C03619=1103.138,282.672,422.520,179.278,15.807,151.492
C03620=1103.132,282.424,422.550,179.274,15.805,151.492
C03621=1103.126,282.176,422.578,179.271,15.805,151.493
C03622=1103.121,281.927,422.607,179.267,15.803,151.493
C03623=1103.115,281.679,422.636,179.264,15.802,151.494
C03624=1103.109,281.431,422.666,179.260,15.801,151.494
C03625=1103.104,281.183,422.695,179.256,15.800,151.495
C03626=1103.098,280.935,422.724,179.252,15.799,151.495
C03627=1103.092,280.687,422.753,179.249,15.798,151.496
C03628=1103.087,280.438,422.782,179.245,15.797,151.496
C03629=1103.081,280.190,422.811,179.242,15.796,151.497
C03630=1103.076,279.942,422.841,179.238,15.795,151.497
C03631=1103.069,279.694,422.870,179.235,15.794,151.498
C03632=1103.064,279.446,422.899,179.231,15.793,151.498
C03633=1103.059,279.197,422.927,179.227,15.792,151.499
C03634=1103.053,278.949,422.957,179.224,15.791,151.499
C03635=1103.047,278.701,422.986,179.220,15.790,151.500
C03636=1103.041,278.453,423.014,179.216,15.789,151.500
C03637=1103.036,278.204,423.044,179.212,15.788,151.501
C03638=1103.030,277.956,423.073,179.209,15.787,151.502
C03639=1103.025,277.708,423.101,179.205,15.786,151.502
C03640=1103.019,277.460,423.130,179.202,15.785,151.503
C03641=1103.013,277.211,423.159,179.198,15.784,151.503
C03642=1103.008,276.963,423.188,179.195,15.783,151.504
C03643=1103.000,276.606,423.229,179.189,15.782,151.504
C03644=1102.991,276.250,423.271,179.184,15.781,151.505
C03645=1102.984,275.893,423.312,179.179,15.780,151.506
C03646=1102.975,275.536,423.353,179.174,15.778,151.507
C03647=1102.969,275.288,423.382,179.170,15.777,151.507
C03648=1102.964,275.039,423.411,179.167,15.776,151.508
C03649=1102.958,274.791,423.440,179.163,15.775,151.508
C03650=1102.952,274.543,423.468,179.159,15.774,151.509
C03651=1102.946,274.294,423.497,179.155,15.773,151.509
C03652=1102.941,274.046,423.526,179.152,15.772,151.510
C03653=1102.935,273.797,423.554,179.148,15.771,151.511
C03654=1102.930,273.550,423.583,179.145,15.770,151.511
C03655=1102.924,273.301,423.611,179.141,15.769,151.512
C03656=1102.918,273.053,423.641,179.138,15.769,151.512
C03657=1102.913,272.805,423.669,179.134,15.767,151.513
C03658=1102.907,272.556,423.697,179.130,15.767,151.513
C03659=1102.901,272.308,423.726,179.127,15.766,151.514
C03660=1102.896,272.060,423.754,179.123,15.765,151.515
C03661=1102.891,271.811,423.783,179.120,15.764,151.515
C03662=1102.885,271.563,423.812,179.116,15.763,151.516
C03663=1102.879,271.314,423.840,179.112,15.762,151.516
C03664=1102.873,271.066,423.868,179.108,15.762,151.517
C03665=1102.867,270.818,423.897,179.105,15.761,151.517
C03666=1102.862,270.570,423.925,179.101,15.760,151.518
C03667=1102.856,270.321,423.953,179.098,15.759,151.518
C03668=1102.851,270.073,423.981,179.094,15.758,151.519
C03669=1102.845,269.825,424.011,179.090,15.757,151.520
C03670=1102.840,269.577,424.039,179.086,15.756,151.520
C03671=1102.834,269.328,424.067,179.083,15.756,151.521
C03672=1102.828,269.079,424.096,179.080,15.755,151.521
C03673=1102.822,268.831,424.124,179.076,15.754,151.522
C03674=1102.816,268.583,424.152,179.072,15.753,151.522
C03675=1102.811,268.335,424.181,179.068,15.752,151.523
C03676=1102.805,268.086,424.209,179.065,15.751,151.524
C03677=1102.800,267.838,424.237,179.061,15.750,151.524
C03678=1102.794,267.590,424.265,179.057,15.750,151.525
C03679=1102.788,267.342,424.293,179.054,15.749,151.525
C03680=1102.782,267.093,424.321,179.050,15.748,151.526
C03681=1102.777,266.845,424.349,179.047,15.748,151.527
C03682=1102.771,266.596,424.378,179.043,15.746,151.527
C03683=1102.766,266.348,424.406,179.040,15.746,151.528
C03684=1102.760,266.100,424.434,179.035,15.745,151.528
C03685=1102.754,265.851,424.462,179.032,15.744,151.529
C03686=1102.749,265.603,424.490,179.028,15.743,151.529
C03687=1102.743,265.354,424.518,179.025,15.743,151.530
C03688=1102.738,265.106,424.546,179.021,15.742,151.531
C03689=1102.732,264.858,424.575,179.017,15.741,151.531
C03690=1102.726,264.610,424.602,179.014,15.740,151.532
C03691=1102.720,264.362,424.630,179.010,15.739,151.532
C03692=1102.714,264.113,424.658,179.006,15.739,151.533
C03693=1102.709,263.865,424.686,179.003,15.738,151.534
C03694=1102.703,263.616,424.714,178.999,15.737,151.534
C03695=1102.695,263.263,424.754,178.994,15.736,151.535
C03696=1102.686,262.908,424.793,178.988,15.735,151.536
C03697=1102.679,262.554,424.833,178.984,15.735,151.537
C03698=1102.670,262.200,424.873,178.978,15.733,151.538
C03699=1102.665,261.952,424.901,178.974,15.732,151.538
C03700=1102.659,261.703,424.929,178.971,15.732,151.539
C03701=1102.653,261.455,424.956,178.968,15.731,151.539
C03702=1102.647,261.206,424.984,178.963,15.730,151.540
C03703=1102.642,260.958,425.012,178.960,15.730,151.541
C03704=1102.636,260.710,425.040,178.956,15.729,151.541
C03705=1102.630,260.461,425.067,178.953,15.728,151.542
C03706=1102.625,260.213,425.095,178.949,15.728,151.543
C03707=1102.618,259.964,425.123,178.945,15.727,151.543
C03708=1102.613,259.716,425.150,178.941,15.726,151.544
C03709=1102.608,259.468,425.178,178.938,15.726,151.544
C03710=1102.601,259.219,425.206,178.934,15.725,151.545
C03711=1102.596,258.971,425.233,178.931,15.724,151.546
C03712=1102.591,258.723,425.261,178.926,15.723,151.546
C03713=1102.584,258.474,425.289,178.923,15.723,151.547
C03714=1102.579,258.225,425.316,178.920,15.722,151.548
C03715=1102.573,257.977,425.344,178.915,15.721,151.548
C03716=1102.567,257.728,425.371,178.912,15.721,151.549
C03717=1102.562,257.480,425.399,178.909,15.721,151.549
C03718=1102.556,257.233,425.426,178.905,15.719,151.550
C03719=1102.550,256.983,425.454,178.901,15.719,151.551
C03720=1102.545,256.735,425.482,178.898,15.718,151.551
C03721=1102.539,256.487,425.509,178.894,15.717,151.552
C03722=1102.533,256.238,425.537,178.890,15.717,151.552
C03723=1102.527,255.990,425.564,178.886,15.716,151.553
C03724=1102.522,255.742,425.591,178.883,15.715,151.554
C03725=1102.517,255.493,425.619,178.879,15.715,151.554
C03726=1102.510,255.244,425.646,178.875,15.714,151.555
C03727=1102.505,254.996,425.674,178.872,15.714,151.556
C03728=1102.499,254.747,425.700,178.868,15.713,151.556
C03729=1102.494,254.499,425.728,178.864,15.712,151.557
C03730=1102.488,254.250,425.755,178.861,15.712,151.558
C03731=1102.483,254.002,425.783,178.858,15.711,151.558
C03732=1102.476,253.754,425.810,178.853,15.710,151.559
C03733=1102.471,253.505,425.837,178.850,15.710,151.559
C03734=1102.465,253.257,425.865,178.847,15.709,151.560
C03735=1102.460,253.008,425.892,178.843,15.708,151.561
C03736=1102.454,252.760,425.919,178.839,15.708,151.561
C03737=1102.449,252.511,425.946,178.835,15.707,151.562
C03738=1102.443,252.263,425.973,178.832,15.706,151.562
C03739=1102.438,252.015,426.001,178.828,15.706,151.563
C03740=1102.431,251.766,426.028,178.824,15.705,151.564
C03741=1102.426,251.517,426.055,178.821,15.705,151.564
C03742=1102.420,251.269,426.082,178.817,15.704,151.565
C03743=1102.415,251.021,426.109,178.813,15.703,151.566
C03744=1102.410,250.772,426.136,178.810,15.702,151.566
C03745=1102.404,250.524,426.163,178.806,15.702,151.567
C03746=1102.398,250.274,426.190,178.802,15.701,151.568
C03747=1102.390,249.918,426.230,178.797,15.701,151.568
C03748=1102.382,249.561,426.268,178.792,15.700,151.569
C03749=1102.374,249.204,426.307,178.787,15.699,151.570
C03750=1102.366,248.847,426.347,178.781,15.698,151.571
C03751=1102.361,248.599,426.373,178.778,15.697,151.572
C03752=1102.355,248.351,426.400,178.775,15.697,151.572
C03753=1102.350,248.102,426.427,178.770,15.696,151.573
C03754=1102.344,247.854,426.454,178.767,15.695,151.574
C03755=1102.339,247.605,426.481,178.764,15.695,151.574
C03756=1102.333,247.357,426.508,178.760,15.694,151.575
C03757=1102.327,247.108,426.534,178.756,15.694,151.575
C03758=1102.322,246.860,426.561,178.753,15.693,151.576
C03759=1102.317,246.611,426.588,178.749,15.692,151.577
C03760=1102.311,246.363,426.615,178.745,15.692,151.577
C03761=1102.304,246.114,426.642,178.741,15.692,151.578
C03762=1102.299,245.865,426.668,178.738,15.691,151.579
C03763=1102.294,245.617,426.696,178.734,15.690,151.579
C03764=1102.288,245.368,426.722,178.730,15.690,151.580
C03765=1102.282,245.120,426.749,178.727,15.689,151.581
C03766=1102.276,244.872,426.776,178.723,15.688,151.581
C03767=1102.272,244.622,426.802,178.719,15.688,151.582
C03768=1102.266,244.374,426.829,178.716,15.688,151.583
C03769=1102.260,244.126,426.855,178.713,15.687,151.583
C03770=1102.254,243.877,426.882,178.708,15.687,151.584
C03771=1102.248,243.629,426.909,178.705,15.686,151.584
C03772=1102.243,243.381,426.935,178.702,15.686,151.585
C03773=1102.238,243.131,426.962,178.697,15.685,151.586
C03774=1102.232,242.883,426.989,178.694,15.684,151.586
C03775=1102.226,242.635,427.015,178.691,15.684,151.587
C03776=1102.221,242.386,427.042,178.687,15.684,151.588
C03777=1102.215,242.138,427.069,178.683,15.683,151.589
C03778=1102.209,241.889,427.094,178.680,15.682,151.589
C03779=1102.204,241.641,427.121,178.676,15.682,151.590
C03780=1102.198,241.392,427.148,178.672,15.681,151.590
C03781=1102.192,241.144,427.174,178.668,15.681,151.591
C03782=1102.187,240.895,427.200,178.665,15.681,151.592
C03783=1102.181,240.646,427.227,178.661,15.680,151.592
C03784=1102.175,240.398,427.254,178.657,15.679,151.593
C03785=1102.170,240.149,427.280,178.654,15.679,151.594
C03786=1102.164,239.901,427.306,178.650,15.679,151.595
C03787=1102.158,239.652,427.333,178.647,15.678,151.595
C03788=1102.153,239.403,427.359,178.642,15.677,151.596
C03789=1102.147,239.155,427.385,178.639,15.677,151.597
C03790=1102.141,238.906,427.411,178.635,15.677,151.597
C03791=1102.136,238.658,427.438,178.632,15.676,151.598
C03792=1102.130,238.409,427.465,178.628,15.676,151.598
C03793=1102.124,238.160,427.491,178.624,15.675,151.599
C03794=1102.119,237.912,427.517,178.621,15.675,151.600
C03795=1102.113,237.663,427.543,178.617,15.675,151.601
C03796=1102.107,237.415,427.569,178.613,15.674,151.601
C03797=1102.101,237.166,427.595,178.610,15.674,151.602
C03798=1102.095,236.918,427.622,178.606,15.673,151.603
C03799=1102.088,236.554,427.660,178.601,15.672,151.603
C03800=1102.079,236.190,427.698,178.595,15.672,151.604
C03801=1102.071,235.827,427.737,178.591,15.671,151.605
C03802=1102.063,235.463,427.774,178.585,15.671,151.606
C03803=1102.057,235.214,427.801,178.581,15.670,151.607
C03804=1102.052,234.965,427.827,178.578,15.670,151.608
C03805=1102.046,234.718,427.853,178.574,15.669,151.608
C03806=1102.041,234.469,427.879,178.570,15.669,151.609
C03807=1102.035,234.220,427.905,178.567,15.669,151.610
C03808=1102.029,233.972,427.931,178.563,15.668,151.610
C03809=1102.023,233.723,427.957,178.559,15.667,151.611
C03810=1102.018,233.474,427.983,178.556,15.667,151.612
C03811=1102.013,233.226,428.009,178.552,15.667,151.612
C03812=1102.007,232.977,428.034,178.549,15.667,151.613
C03813=1102.001,232.728,428.060,178.545,15.666,151.614
C03814=1101.996,232.479,428.086,178.541,15.666,151.615
C03815=1101.990,232.231,428.113,178.538,15.665,151.615
C03816=1101.984,231.982,428.138,178.534,15.665,151.616
C03817=1101.979,231.734,428.164,178.530,15.665,151.617
C03818=1101.973,231.485,428.190,178.526,15.664,151.617
C03819=1101.968,231.237,428.216,178.523,15.663,151.618
C03820=1101.961,230.988,428.242,178.519,15.663,151.619
C03821=1101.956,230.739,428.268,178.516,15.663,151.619
C03822=1101.951,230.491,428.293,178.512,15.662,151.620
C03823=1101.945,230.242,428.319,178.508,15.662,151.621
C03824=1101.939,229.993,428.345,178.505,15.661,151.621
C03825=1101.933,229.745,428.371,178.501,15.661,151.622
C03826=1101.927,229.496,428.397,178.497,15.661,151.623
C03827=1101.923,229.248,428.422,178.494,15.661,151.623
C03828=1101.916,228.999,428.447,178.491,15.660,151.624
C03829=1101.911,228.750,428.473,178.486,15.659,151.625
C03830=1101.905,228.502,428.499,178.483,15.659,151.625
C03831=1101.900,228.253,428.524,178.479,15.659,151.626
C03832=1101.894,228.005,428.550,178.476,15.659,151.627
C03833=1101.888,227.756,428.576,178.472,15.659,151.628
C03834=1101.882,227.507,428.601,178.468,15.658,151.628
C03835=1101.877,227.259,428.626,178.464,15.658,151.629
C03836=1101.872,227.010,428.652,178.461,15.658,151.630
C03837=1101.865,226.761,428.678,178.458,15.657,151.630
C03838=1101.860,226.512,428.704,178.454,15.657,151.631
C03839=1101.854,226.264,428.729,178.451,15.657,151.632
C03840=1101.849,226.015,428.755,178.446,15.656,151.632
C03841=1101.843,225.766,428.780,178.443,15.656,151.633
C03842=1101.838,225.518,428.806,178.439,15.655,151.634
C03843=1101.832,225.269,428.831,178.436,15.655,151.635
C03844=1101.826,225.020,428.857,178.432,15.655,151.635
C03845=1101.820,224.772,428.882,178.429,15.654,151.636
C03846=1101.815,224.523,428.906,178.425,15.654,151.636
C03847=1101.809,224.274,428.932,178.421,15.653,151.637
C03848=1101.803,224.026,428.958,178.417,15.653,151.638
C03849=1101.798,223.777,428.983,178.414,15.653,151.639
C03850=1101.792,223.529,429.009,178.410,15.653,151.639
C03851=1101.784,223.156,429.046,178.405,15.652,151.640
C03852=1101.776,222.784,429.084,178.399,15.651,151.641
C03853=1101.767,222.412,429.122,178.394,15.651,151.642
C03854=1101.759,222.040,429.160,178.389,15.651,151.643
C03855=1101.753,221.792,429.185,178.385,15.651,151.644
C03856=1101.747,221.543,429.210,178.382,15.650,151.645
C03857=1101.741,221.294,429.236,178.377,15.650,151.646
C03858=1101.737,221.045,429.260,178.374,15.649,151.646
C03859=1101.730,220.797,429.286,178.370,15.649,151.647
C03860=1101.724,220.548,429.311,178.367,15.649,151.648
C03861=1101.719,220.299,429.335,178.363,15.649,151.648
C03862=1101.713,220.050,429.361,178.360,15.649,151.649
C03863=1101.707,219.802,429.387,178.356,15.649,151.650
C03864=1101.702,219.553,429.411,178.352,15.648,151.651
C03865=1101.696,219.304,429.436,178.349,15.647,151.651
C03866=1101.691,219.056,429.461,178.345,15.647,151.652
C03867=1101.685,218.807,429.486,178.341,15.647,151.653
C03868=1101.679,218.559,429.511,178.338,15.647,151.653
C03869=1101.673,218.310,429.536,178.334,15.647,151.654
C03870=1101.668,218.061,429.562,178.331,15.646,151.655
C03871=1101.663,217.812,429.586,178.327,15.646,151.655
C03872=1101.656,217.563,429.612,178.323,15.645,151.656
C03873=1101.651,217.315,429.636,178.319,15.645,151.657
C03874=1101.645,217.066,429.661,178.316,15.645,151.658
C03875=1101.640,216.817,429.686,178.312,15.645,151.658
C03876=1101.634,216.569,429.711,178.309,15.645,151.659
C03877=1101.629,216.320,429.736,178.305,15.645,151.660
C03878=1101.623,216.071,429.761,178.302,15.644,151.660
C03879=1101.617,215.823,429.785,178.298,15.644,151.661
C03880=1101.611,215.574,429.811,178.295,15.644,151.662
C03881=1101.606,215.326,429.835,178.291,15.643,151.662
C03882=1101.601,215.076,429.860,178.287,15.643,151.663
C03883=1101.595,214.828,429.885,178.284,15.643,151.664
C03884=1101.589,214.579,429.910,178.280,15.642,151.665
C03885=1101.584,214.331,429.935,178.276,15.642,151.665
C03886=1101.578,214.081,429.959,178.273,15.642,151.666
C03887=1101.572,213.833,429.983,178.269,15.642,151.667
C03888=1101.567,213.585,430.008,178.266,15.642,151.667
C03889=1101.561,213.336,430.033,178.262,15.642,151.668
C03890=1101.556,213.087,430.057,178.258,15.641,151.669
C03891=1101.550,212.838,430.082,178.254,15.641,151.670
C03892=1101.544,212.590,430.107,178.251,15.641,151.670
C03893=1101.538,212.340,430.131,178.247,15.640,151.671
C03894=1101.533,212.092,430.156,178.244,15.640,151.672
C03895=1101.527,211.843,430.181,178.240,15.640,151.672
C03896=1101.521,211.595,430.205,178.237,15.640,151.673
C03897=1101.516,211.346,430.230,178.233,15.640,151.674
C03898=1101.510,211.097,430.254,178.230,15.639,151.674
C03899=1101.505,210.848,430.278,178.226,15.639,151.675
C03900=1101.499,210.599,430.304,178.223,15.639,151.676
C03901=1101.493,210.351,430.328,178.218,15.638,151.677
C03902=1101.487,210.102,430.353,178.215,15.638,151.677
C03903=1101.480,209.733,430.389,178.210,15.638,151.678
C03904=1101.471,209.366,430.425,178.204,15.637,151.679
C03905=1101.463,208.997,430.461,178.199,15.638,151.680
C03906=1101.455,208.628,430.497,178.194,15.637,151.682
C03907=1101.431,207.624,430.595,178.158,15.629,151.687
C03908=1101.426,207.375,430.619,178.154,15.629,151.688
C03909=1101.420,207.126,430.644,178.150,15.630,151.689
C03910=1101.414,206.878,430.668,178.146,15.630,151.690
C03911=1101.409,206.629,430.692,178.143,15.631,151.691
C03912=1101.403,206.380,430.717,178.139,15.632,151.692
C03913=1101.397,206.132,430.740,178.135,15.632,151.693
C03914=1101.392,205.882,430.764,178.131,15.633,151.694
C03915=1101.387,205.634,430.788,178.128,15.634,151.695
C03916=1101.381,205.384,430.813,178.124,15.634,151.696
C03917=1101.375,205.136,430.836,178.120,15.635,151.697
C03918=1101.369,204.888,430.861,178.116,15.635,151.698
C03919=1101.363,204.638,430.885,178.112,15.636,151.699
C03920=1101.357,204.390,430.909,178.109,15.637,151.700
C03921=1101.352,204.141,430.932,178.105,15.637,151.700
C03922=1101.347,203.892,430.957,178.100,15.638,151.701
C03923=1101.340,203.643,430.981,178.097,15.638,151.702
C03924=1101.335,203.395,431.005,178.094,15.639,151.703
C03925=1101.330,203.145,431.028,178.089,15.640,151.704
C03926=1101.324,202.897,431.052,178.086,15.640,151.705
C03927=1101.319,202.649,431.076,178.082,15.641,151.706
C03928=1101.312,202.400,431.100,178.077,15.641,151.707
C03929=1101.307,202.150,431.124,178.074,15.642,151.708
C03930=1101.301,201.902,431.148,178.070,15.643,151.709
C03931=1101.295,201.653,431.172,178.066,15.643,151.710
C03932=1101.289,201.405,431.196,178.063,15.644,151.711
C03933=1101.284,201.155,431.219,178.059,15.645,151.712
C03934=1101.278,200.907,431.243,178.055,15.645,151.713
C03935=1101.272,200.658,431.268,178.051,15.646,151.714
C03936=1101.267,200.409,431.291,178.047,15.646,151.715
C03937=1101.260,200.161,431.314,178.044,15.647,151.715
C03938=1101.255,199.911,431.338,178.040,15.648,151.717
C03939=1101.249,199.662,431.362,178.036,15.649,151.717
C03940=1101.244,199.414,431.386,178.032,15.649,151.718
C03941=1101.238,199.165,431.409,178.029,15.650,151.719
C03942=1101.233,198.916,431.433,178.025,15.651,151.720
C03943=1101.227,198.668,431.456,178.021,15.651,151.721
C03944=1101.220,198.419,431.480,178.017,15.652,151.722
C03945=1101.215,198.169,431.504,178.014,15.653,151.723
C03946=1101.209,197.921,431.527,178.010,15.653,151.724
C03947=1101.204,197.672,431.551,178.006,15.654,151.725
C03948=1101.198,197.424,431.575,178.002,15.654,151.726
C03949=1101.192,197.175,431.598,177.999,15.655,151.727
C03950=1101.187,196.926,431.622,177.995,15.656,151.728
C03951=1101.181,196.676,431.645,177.991,15.656,151.729
C03952=1101.175,196.428,431.669,177.987,15.656,151.729
C03953=1101.170,196.179,431.692,177.984,15.657,151.730
C03954=1101.164,195.931,431.716,177.980,15.658,151.731
C03955=1101.159,195.682,431.740,177.976,15.658,151.732
C03956=1101.153,195.433,431.763,177.972,15.659,151.733
C03957=1101.147,195.184,431.786,177.969,15.660,151.734
C03958=1101.142,194.935,431.810,177.965,15.660,151.735
C03959=1101.135,194.686,431.834,177.961,15.661,151.736
C03960=1101.130,194.437,431.857,177.957,15.661,151.737
C03961=1101.124,194.188,431.880,177.954,15.662,151.738
C03962=1101.119,193.940,431.904,177.950,15.662,151.739
C03963=1101.113,193.691,431.927,177.946,15.663,151.739
C03964=1101.107,193.442,431.950,177.942,15.663,151.741
C03965=1101.102,193.193,431.974,177.939,15.664,151.741
C03966=1101.096,192.944,431.997,177.935,15.665,151.742
C03967=1101.090,192.696,432.020,177.931,15.665,151.743
C03968=1101.084,192.423,432.046,177.927,15.666,151.744
C03969=1101.079,192.150,432.071,177.923,15.666,151.745
C03970=1101.071,191.877,432.097,177.919,15.667,151.746
C03971=1101.066,191.604,432.122,177.915,15.667,151.747
C03972=1101.059,191.356,432.146,177.911,15.668,151.748
C03973=1101.054,191.107,432.169,177.908,15.669,151.749
C03974=1101.049,190.858,432.192,177.904,15.669,151.750
C03975=1101.043,190.609,432.215,177.900,15.670,151.751
C03976=1101.037,190.360,432.238,177.896,15.670,151.752
C03977=1101.032,190.112,432.262,177.893,15.671,151.753
C03978=1101.026,189.863,432.285,177.889,15.671,151.753
C03979=1101.021,189.614,432.308,177.886,15.672,151.754
C03980=1101.015,189.365,432.331,177.882,15.672,151.755
C03981=1101.010,189.116,432.355,177.879,15.673,151.756
C03982=1101.005,188.868,432.377,177.875,15.673,151.757
C03983=1100.999,188.619,432.400,177.871,15.674,151.758
C03984=1100.993,188.370,432.423,177.867,15.674,151.759
C03985=1100.987,188.121,432.446,177.864,15.675,151.760
C03986=1100.982,187.872,432.469,177.860,15.675,151.760
C03987=1100.977,187.623,432.493,177.856,15.676,151.761
C03988=1100.971,187.374,432.516,177.852,15.676,151.762
C03989=1100.965,187.125,432.539,177.849,15.677,151.763
C03990=1100.959,186.877,432.562,177.845,15.677,151.764
C03991=1100.954,186.627,432.585,177.841,15.678,151.765
C03992=1100.948,186.378,432.607,177.838,15.677,151.766
C03993=1100.943,186.129,432.631,177.835,15.678,151.766
C03994=1100.938,185.881,432.654,177.831,15.679,151.767
C03995=1100.932,185.632,432.677,177.827,15.679,151.768
C03996=1100.927,185.383,432.699,177.824,15.680,151.769
C03997=1100.921,185.134,432.722,177.820,15.680,151.770
C03998=1100.915,184.885,432.745,177.816,15.681,151.771
C03999=1100.909,184.636,432.768,177.812,15.681,151.772
C04000=1100.904,184.387,432.791,177.809,15.682,151.773
C04001=1100.898,184.139,432.814,177.805,15.682,151.774
C04002=1100.891,183.890,432.837,177.802,15.683,151.774
C04003=1100.886,183.641,432.859,177.799,15.684,151.775
C04004=1100.880,183.392,432.882,177.795,15.684,151.776
C04005=1100.875,183.143,432.905,177.791,15.684,151.777
C04006=1100.869,182.894,432.928,177.787,15.685,151.778
C04007=1100.863,182.645,432.951,177.784,15.686,151.779
C04008=1100.857,182.396,432.973,177.780,15.686,151.780
C04009=1100.851,182.147,432.996,177.776,15.687,151.781
C04010=1100.846,181.899,433.018,177.773,15.688,151.781
C04011=1100.840,181.650,433.041,177.769,15.688,151.782
C04012=1100.835,181.401,433.064,177.765,15.688,151.783
C04013=1100.829,181.152,433.087,177.761,15.689,151.784
C04014=1100.822,180.903,433.109,177.758,15.690,151.785
C04015=1100.817,180.654,433.131,177.754,15.690,151.786
C04016=1100.811,180.405,433.154,177.751,15.690,151.787
C04017=1100.805,180.156,433.177,177.748,15.691,151.788
C04018=1100.799,179.907,433.199,177.744,15.692,151.789
C04019=1100.794,179.659,433.221,177.740,15.692,151.789
C04020=1100.788,179.410,433.244,177.737,15.693,151.790
C04021=1100.783,179.161,433.267,177.733,15.693,151.791
C04022=1100.777,178.912,433.289,177.729,15.693,151.792
C04023=1100.771,178.663,433.312,177.725,15.694,151.793
C04024=1100.765,178.414,433.335,177.722,15.695,151.794
C04025=1100.760,178.164,433.357,177.718,15.695,151.795
C04026=1100.754,177.916,433.379,177.715,15.695,151.796
C04027=1100.748,177.667,433.401,177.712,15.696,151.796
C04028=1100.743,177.418,433.424,177.708,15.696,151.797
C04029=1100.737,177.169,433.447,177.704,15.697,151.798
C04030=1100.731,176.920,433.469,177.701,15.698,151.799
C04031=1100.726,176.672,433.491,177.697,15.698,151.800
C04032=1100.719,176.399,433.516,177.693,15.698,151.801
C04033=1100.712,176.125,433.540,177.689,15.699,151.802
C04034=1100.707,175.852,433.565,177.686,15.699,151.802
C04035=1100.701,175.579,433.589,177.681,15.700,151.803
C04036=1100.695,175.331,433.611,177.678,15.700,151.804
C04037=1100.689,175.081,433.634,177.675,15.701,151.805
C04038=1100.684,174.832,433.656,177.671,15.701,151.806
C04039=1100.677,174.583,433.678,177.667,15.702,151.807
C04040=1100.672,174.335,433.701,177.664,15.702,151.808
C04041=1100.667,174.085,433.723,177.660,15.702,151.808
C04042=1100.661,173.836,433.745,177.656,15.703,151.809
C04043=1100.655,173.587,433.768,177.653,15.703,151.810
C04044=1100.650,173.338,433.789,177.650,15.704,151.811
C04045=1100.644,173.090,433.812,177.646,15.704,151.812
C04046=1100.638,172.840,433.834,177.642,15.704,151.813
C04047=1100.633,172.592,433.856,177.639,15.705,151.813
C04048=1100.627,172.343,433.878,177.635,15.705,151.814
C04049=1100.622,172.093,433.900,177.632,15.705,151.815
C04050=1100.616,171.846,433.922,177.629,15.706,151.816
C04051=1100.610,171.596,433.945,177.625,15.706,151.817
C04052=1100.605,171.347,433.967,177.621,15.707,151.818
C04053=1100.599,171.098,433.988,177.618,15.708,151.818
C04054=1100.594,170.849,434.011,177.615,15.708,151.819
C04055=1100.587,170.600,434.033,177.611,15.708,151.820
C04056=1100.583,170.351,434.055,177.607,15.708,151.821
C04057=1100.577,170.102,434.078,177.604,15.709,151.822
C04058=1100.571,169.853,434.099,177.601,15.709,151.822
C04059=1100.566,169.604,434.121,177.597,15.709,151.823
C04060=1100.560,169.355,434.143,177.594,15.710,151.824
C04061=1100.555,169.107,434.165,177.590,15.710,151.825
C04062=1100.548,168.858,434.187,177.587,15.710,151.826
C04063=1100.543,168.608,434.209,177.583,15.711,151.827
C04064=1100.537,168.360,434.230,177.580,15.711,151.827
C04065=1100.532,168.110,434.253,177.576,15.711,151.828
C04066=1100.526,167.862,434.274,177.573,15.712,151.829
C04067=1100.521,167.613,434.297,177.569,15.712,151.830
C04068=1100.515,167.363,434.319,177.566,15.712,151.830
C04069=1100.510,167.115,434.340,177.563,15.713,151.831
C04070=1100.504,166.865,434.363,177.559,15.713,151.832
C04071=1100.499,166.617,434.384,177.555,15.714,151.833
C04072=1100.493,166.367,434.406,177.552,15.714,151.834
C04073=1100.488,166.119,434.427,177.549,15.714,151.834
C04074=1100.482,165.869,434.450,177.545,15.714,151.835
C04075=1100.477,165.621,434.471,177.542,15.714,151.836
C04076=1100.471,165.371,434.492,177.539,15.715,151.837
C04077=1100.465,165.123,434.515,177.535,15.715,151.838
C04078=1100.459,164.874,434.537,177.531,15.715,151.838
C04079=1100.454,164.625,434.559,177.528,15.716,151.839
C04080=1100.448,164.376,434.580,177.525,15.716,151.840
C04081=1100.443,164.127,434.602,177.521,15.716,151.841
C04082=1100.437,163.878,434.624,177.518,15.717,151.842
C04083=1100.433,163.628,434.645,177.514,15.717,151.842
C04084=1100.427,163.379,434.666,177.511,15.717,151.843
C04085=1100.422,163.130,434.688,177.508,15.718,151.844
C04086=1100.416,162.881,434.710,177.504,15.718,151.845
C04087=1100.410,162.633,434.731,177.501,15.718,151.845
C04088=1100.405,162.383,434.753,177.498,15.719,151.846
C04089=1100.399,162.135,434.775,177.494,15.719,151.847
C04090=1100.394,161.885,434.797,177.490,15.719,151.848
C04091=1100.388,161.637,434.818,177.488,15.719,151.848
C04092=1100.382,161.388,434.840,177.484,15.719,151.849
C04093=1100.376,161.139,434.861,177.480,15.720,151.850
C04094=1100.371,160.889,434.883,177.477,15.720,151.851
C04095=1100.366,160.640,434.904,177.474,15.720,151.852
C04096=1100.359,160.367,434.928,177.470,15.721,151.852
C04097=1100.353,160.094,434.951,177.466,15.721,151.853
C04098=1100.347,159.820,434.975,177.462,15.722,151.854
C04099=1100.341,159.547,434.998,177.459,15.721,151.855
C04100=1100.335,159.298,435.020,177.456,15.723,151.856
C04101=1100.329,159.049,435.041,177.452,15.722,151.857
C04102=1100.324,158.800,435.062,177.448,15.722,151.857
C04103=1100.318,158.550,435.084,177.445,15.723,151.858
C04104=1100.313,158.302,435.105,177.442,15.723,151.859
C04105=1100.307,158.053,435.127,177.438,15.723,151.860
C04106=1100.301,157.804,435.147,177.435,15.724,151.860
C04107=1100.295,157.554,435.169,177.432,15.724,151.861
C04108=1100.290,157.306,435.190,177.428,15.724,151.862
C04109=1100.283,157.057,435.212,177.425,15.725,151.863
C04110=1100.279,156.807,435.233,177.422,15.725,151.863
C04111=1100.273,156.559,435.254,177.418,15.725,151.864
C04112=1100.267,156.309,435.276,177.415,15.726,151.865
C04113=1100.262,156.060,435.297,177.411,15.726,151.866
C04114=1100.256,155.811,435.318,177.408,15.726,151.867
C04115=1100.250,155.563,435.340,177.405,15.726,151.867
C04116=1100.245,155.314,435.360,177.402,15.726,151.868
C04117=1100.239,155.064,435.382,177.398,15.727,151.869
C04118=1100.233,154.815,435.402,177.395,15.727,151.870
C04119=1100.227,154.566,435.424,177.391,15.727,151.870
C04120=1100.222,154.317,435.445,177.389,15.728,151.871
C04121=1100.217,154.068,435.466,177.385,15.728,151.872
C04122=1100.210,153.819,435.487,177.381,15.728,151.873
C04123=1100.205,153.570,435.508,177.379,15.728,151.873
C04124=1100.199,153.321,435.530,177.375,15.729,151.874
C04125=1100.194,153.072,435.550,177.371,15.729,151.875
C04126=1100.188,152.823,435.571,177.368,15.729,151.876
C04127=1100.182,152.573,435.592,177.365,15.729,151.876
C04128=1100.177,152.325,435.614,177.361,15.729,151.877
C04129=1100.171,152.076,435.634,177.359,15.730,151.878
C04130=1100.165,151.827,435.656,177.355,15.730,151.879
C04131=1100.160,151.577,435.676,177.352,15.730,151.879
C04132=1100.154,151.329,435.698,177.349,15.730,151.880
C04133=1100.149,151.079,435.718,177.345,15.730,151.881
C04134=1100.143,150.831,435.740,177.342,15.731,151.881
C04135=1100.138,150.581,435.760,177.339,15.731,151.882
C04136=1100.132,150.332,435.782,177.335,15.731,151.883
C04137=1100.126,150.083,435.803,177.332,15.731,151.884
C04138=1100.121,149.834,435.823,177.329,15.731,151.884
C04139=1100.115,149.586,435.844,177.325,15.731,151.885
C04140=1100.109,149.336,435.865,177.322,15.732,151.886
C04141=1100.103,149.087,435.886,177.319,15.732,151.887
C04142=1100.098,148.838,435.906,177.316,15.732,151.887
C04143=1100.092,148.589,435.927,177.313,15.732,151.888
C04144=1100.087,148.340,435.949,177.309,15.732,151.889
C04145=1100.081,148.091,435.969,177.306,15.733,151.889
C04146=1100.075,147.841,435.990,177.303,15.733,151.890
C04147=1100.069,147.593,436.011,177.299,15.733,151.891
C04148=1100.064,147.344,436.031,177.296,15.733,151.892
C04149=1100.059,147.095,436.052,177.293,15.733,151.892
C04150=1100.053,146.845,436.073,177.289,15.733,151.893
C04151=1100.047,146.597,436.094,177.286,15.734,151.894
C04152=1100.041,146.347,436.114,177.283,15.734,151.895
C04153=1100.036,146.098,436.135,177.280,15.735,151.895
C04154=1100.030,145.849,436.156,177.276,15.735,151.896
C04155=1100.024,145.600,436.176,177.273,15.734,151.897
C04156=1100.019,145.351,436.197,177.270,15.735,151.898
C04157=1100.013,145.102,436.217,177.266,15.735,151.898
C04158=1100.008,144.852,436.238,177.263,15.735,151.899
C04159=1100.002,144.603,436.258,177.260,15.735,151.900
C04160=1099.996,144.330,436.282,177.257,15.736,151.900
C04161=1099.989,144.056,436.304,177.253,15.736,151.901
C04162=1099.983,143.783,436.326,177.249,15.736,151.902
C04163=1099.977,143.509,436.349,177.246,15.736,151.903
C04164=1099.971,143.260,436.369,177.243,15.736,151.903
C04165=1099.966,143.010,436.390,177.240,15.736,151.904
C04166=1099.960,142.762,436.410,177.236,15.736,151.905
C04167=1099.954,142.512,436.431,177.233,15.737,151.906
C04168=1099.949,142.263,436.451,177.230,15.736,151.906
C04169=1099.944,142.014,436.472,177.227,15.737,151.907
C04170=1099.938,141.765,436.492,177.224,15.737,151.908
C04171=1099.932,141.515,436.513,177.220,15.737,151.908
C04172=1099.927,141.266,436.533,177.218,15.737,151.909
C04173=1099.921,141.018,436.553,177.214,15.737,151.910
C04174=1099.915,140.769,436.575,177.211,15.737,151.910
C04175=1099.909,140.520,436.595,177.208,15.737,151.911
C04176=1099.904,140.271,436.615,177.204,15.737,151.912
C04177=1099.899,140.022,436.636,177.202,15.738,151.912
C04178=1099.892,139.772,436.655,177.198,15.738,151.913
C04179=1099.887,139.523,436.676,177.194,15.738,151.914
C04180=1099.881,139.274,436.696,177.192,15.738,151.914
C04181=1099.876,139.025,436.716,177.188,15.738,151.915
C04182=1099.870,138.776,436.736,177.186,15.738,151.916
C04183=1099.865,138.527,436.757,177.182,15.738,151.917
C04184=1099.859,138.278,436.777,177.179,15.738,151.917
C04185=1099.853,138.028,436.798,177.176,15.738,151.918
C04186=1099.847,137.779,436.818,177.172,15.738,151.919
C04187=1099.841,137.530,436.838,177.170,15.739,151.919
C04188=1099.835,137.281,436.858,177.166,15.739,151.920
C04189=1099.830,137.032,436.879,177.163,15.739,151.921
C04190=1099.825,136.783,436.898,177.160,15.739,151.921
C04191=1099.819,136.534,436.919,177.157,15.739,151.922
C04192=1099.813,136.285,436.939,177.154,15.739,151.923
C04193=1099.808,136.036,436.959,177.151,15.739,151.923
C04194=1099.802,135.787,436.979,177.147,15.739,151.924
C04195=1099.796,135.537,437.000,177.145,15.739,151.925
C04196=1099.790,135.288,437.019,177.141,15.739,151.925
C04197=1099.785,135.039,437.040,177.138,15.740,151.926
C04198=1099.779,134.790,437.060,177.135,15.739,151.927
C04199=1099.773,134.541,437.080,177.131,15.739,151.927
C04200=1099.768,134.291,437.100,177.129,15.739,151.928
C04201=1099.762,134.042,437.120,177.125,15.739,151.929
C04202=1099.757,133.793,437.140,177.123,15.739,151.929
C04203=1099.751,133.545,437.160,177.119,15.739,151.930
C04204=1099.746,133.295,437.180,177.116,15.739,151.931
C04205=1099.740,133.046,437.200,177.113,15.739,151.931
C04206=1099.734,132.797,437.220,177.110,15.739,151.932
C04207=1099.729,132.547,437.240,177.107,15.740,151.933
C04208=1099.723,132.299,437.260,177.104,15.740,151.933
C04209=1099.717,132.050,437.280,177.100,15.739,151.934
C04210=1099.712,131.800,437.299,177.098,15.740,151.935
C04211=1099.706,131.551,437.319,177.094,15.739,151.935
C04212=1099.700,131.302,437.339,177.092,15.740,151.936
C04213=1099.695,131.053,437.359,177.088,15.739,151.937
C04214=1099.689,130.804,437.379,177.085,15.739,151.937
C04215=1099.683,130.555,437.399,177.082,15.740,151.938
C04216=1099.678,130.306,437.418,177.079,15.740,151.939
C04217=1099.672,130.057,437.438,177.076,15.740,151.939
C04218=1099.666,129.807,437.458,177.073,15.740,151.940
C04219=1099.661,129.558,437.478,177.070,15.740,151.940
C04220=1099.655,129.309,437.498,177.067,15.740,151.941
C04221=1099.649,129.060,437.517,177.063,15.739,151.942
C04222=1099.643,128.811,437.537,177.061,15.740,151.943
C04223=1099.637,128.562,437.556,177.057,15.740,151.943
C04224=1099.631,128.288,437.579,177.054,15.740,151.944
C04225=1099.625,128.013,437.600,177.051,15.740,151.945
C04226=1099.618,127.740,437.622,177.047,15.740,151.945
C04227=1099.612,127.466,437.644,177.044,15.740,151.946
C04228=1099.606,127.217,437.663,177.040,15.740,151.947
C04229=1099.600,126.967,437.682,177.038,15.740,151.947
C04230=1099.595,126.718,437.703,177.034,15.740,151.948
C04231=1099.589,126.469,437.722,177.032,15.740,151.949
C04232=1099.583,126.220,437.742,177.029,15.740,151.949
C04233=1099.578,125.971,437.761,177.025,15.740,151.950
C04234=1099.572,125.723,437.781,177.023,15.740,151.950
C04235=1099.567,125.473,437.800,177.019,15.739,151.951
C04236=1099.561,125.224,437.819,177.017,15.740,151.952
C04237=1099.555,124.975,437.839,177.013,15.740,151.952
C04238=1099.550,124.725,437.859,177.011,15.740,151.953
C04239=1099.544,124.476,437.879,177.007,15.740,151.954
C04240=1099.538,124.227,437.898,177.004,15.739,151.954
C04241=1099.533,123.977,437.918,177.002,15.739,151.955
C04242=1099.527,123.729,437.938,176.998,15.739,151.956
C04243=1099.521,123.479,437.957,176.995,15.740,151.956
C04244=1099.516,123.230,437.976,176.992,15.739,151.957
C04245=1099.510,122.982,437.996,176.990,15.739,151.957
C04246=1099.504,122.732,438.015,176.986,15.739,151.958
C04247=1099.499,122.483,438.034,176.983,15.739,151.959
C04248=1099.493,122.233,438.053,176.980,15.739,151.959
C04249=1099.487,121.985,438.073,176.977,15.739,151.960
C04250=1099.482,121.735,438.093,176.975,15.739,151.960
C04251=1099.477,121.486,438.112,176.971,15.739,151.961
C04252=1099.471,121.237,438.131,176.969,15.739,151.962
C04253=1099.465,120.988,438.151,176.965,15.738,151.962
C04254=1099.460,120.738,438.171,176.962,15.738,151.963
C04255=1099.454,120.489,438.190,176.960,15.738,151.963
C04256=1099.449,120.240,438.209,176.956,15.738,151.964
C04257=1099.443,119.991,438.228,176.954,15.738,151.965
C04258=1099.437,119.741,438.247,176.950,15.738,151.965
C04259=1099.431,119.493,438.267,176.948,15.738,151.966
C04260=1099.426,119.243,438.286,176.944,15.738,151.966
C04261=1099.421,118.994,438.305,176.941,15.737,151.967
C04262=1099.415,118.745,438.324,176.939,15.737,151.967
C04263=1099.409,118.496,438.344,176.935,15.737,151.968
C04264=1099.404,118.246,438.363,176.933,15.737,151.969
C04265=1099.398,117.997,438.382,176.930,15.737,151.969
C04266=1099.393,117.748,438.401,176.927,15.737,151.970
C04267=1099.387,117.499,438.421,176.924,15.736,151.970
C04268=1099.381,117.250,438.440,176.921,15.736,151.971
C04269=1099.376,117.001,438.459,176.918,15.736,151.971
C04270=1099.370,116.752,438.478,176.915,15.736,151.972
C04271=1099.365,116.502,438.498,176.912,15.736,151.973
C04272=1099.359,116.253,438.517,176.909,15.736,151.973
C04273=1099.353,116.004,438.535,176.907,15.735,151.974
C04274=1099.347,115.755,438.554,176.903,15.735,151.974
C04275=1099.342,115.505,438.574,176.901,15.735,151.975
C04276=1099.337,115.257,438.593,176.898,15.735,151.976
C04277=1099.331,115.007,438.612,176.894,15.734,151.976
C04278=1099.325,114.758,438.631,176.892,15.734,151.977
C04279=1099.320,114.509,438.650,176.889,15.734,151.977
C04280=1099.314,114.260,438.669,176.886,15.734,151.978
C04281=1099.309,114.010,438.688,176.883,15.734,151.978
C04282=1099.303,113.760,438.706,176.880,15.734,151.979
C04283=1099.298,113.512,438.725,176.877,15.734,151.980
C04284=1099.292,113.262,438.744,176.875,15.734,151.980
C04285=1099.286,113.013,438.764,176.871,15.733,151.981
C04286=1099.281,112.763,438.783,176.868,15.733,151.981
C04287=1099.275,112.515,438.801,176.866,15.733,151.982
C04288=1099.269,112.241,438.822,176.862,15.733,151.982
C04289=1099.262,111.967,438.843,176.859,15.733,151.983
C04290=1099.256,111.693,438.864,176.856,15.732,151.984
C04291=1099.250,111.420,438.885,176.853,15.732,151.984
C04292=1099.244,111.170,438.903,176.850,15.732,151.985
C04293=1099.239,110.920,438.922,176.847,15.732,151.986
C04294=1099.233,110.672,438.941,176.844,15.732,151.986
C04295=1099.227,110.422,438.960,176.842,15.732,151.987
C04296=1099.222,110.173,438.979,176.838,15.731,151.987
C04297=1099.216,109.925,438.997,176.835,15.731,151.988
C04298=1099.210,109.674,439.016,176.833,15.731,151.988
C04299=1099.204,109.425,439.035,176.830,15.730,151.989
C04300=1099.199,109.177,439.053,176.827,15.730,151.989
C04301=1099.193,108.927,439.073,176.824,15.730,151.990
C04302=1099.187,108.677,439.091,176.821,15.730,151.991
C04303=1099.182,108.429,439.109,176.818,15.730,151.991
C04304=1099.176,108.179,439.129,176.816,15.730,151.992
C04305=1099.170,107.930,439.147,176.812,15.729,151.992
C04306=1099.165,107.681,439.166,176.810,15.729,151.993
C04307=1099.159,107.432,439.184,176.807,15.729,151.993
C04308=1099.153,107.182,439.203,176.804,15.729,151.994
C04309=1099.148,106.933,439.222,176.801,15.728,151.994
C04310=1099.142,106.684,439.240,176.799,15.729,151.995
C04311=1099.137,106.435,439.259,176.796,15.728,151.995
C04312=1099.131,106.185,439.277,176.792,15.727,151.996
C04313=1099.125,105.936,439.296,176.790,15.727,151.997
C04314=1099.119,105.687,439.314,176.787,15.727,151.997
C04315=1099.114,105.437,439.333,176.784,15.727,151.998
C04316=1099.109,105.189,439.352,176.781,15.726,151.998
C04317=1099.102,104.939,439.370,176.779,15.726,151.999
C04318=1099.097,104.690,439.389,176.775,15.726,151.999
C04319=1099.091,104.440,439.407,176.773,15.726,152.000
C04320=1099.086,104.191,439.426,176.770,15.725,152.000
C04321=1099.080,103.943,439.444,176.768,15.726,152.001
C04322=1099.074,103.693,439.463,176.764,15.725,152.001
C04323=1099.068,103.444,439.481,176.762,15.725,152.002
C04324=1099.063,103.194,439.500,176.759,15.724,152.002
C04325=1099.057,102.946,439.518,176.756,15.725,152.003
C04326=1099.052,102.696,439.536,176.753,15.724,152.003
C04327=1099.046,102.447,439.555,176.751,15.724,152.004
C04328=1099.041,102.197,439.573,176.748,15.723,152.004
C04329=1099.035,101.949,439.591,176.745,15.723,152.005
C04330=1099.029,101.699,439.610,176.742,15.723,152.006
C04331=1099.024,101.450,439.628,176.739,15.722,152.006
C04332=1099.018,101.200,439.647,176.737,15.722,152.007
C04333=1099.012,100.950,439.665,176.733,15.722,152.007
C04334=1099.007,100.702,439.684,176.731,15.721,152.008
C04335=1099.001,100.452,439.702,176.728,15.721,152.008
C04336=1098.995,100.204,439.720,176.725,15.721,152.009
C04337=1098.990,99.954,439.738,176.722,15.720,152.009
C04338=1098.984,99.705,439.757,176.720,15.720,152.010
C04339=1098.978,99.455,439.775,176.717,15.720,152.010
C04340=1098.973,99.206,439.793,176.715,15.720,152.011
C04341=1098.967,98.957,439.811,176.711,15.719,152.011
C04342=1098.961,98.708,439.829,176.709,15.719,152.012
C04343=1098.956,98.458,439.847,176.706,15.719,152.012
C04344=1098.950,98.209,439.866,176.703,15.719,152.013
C04345=1098.944,97.960,439.884,176.700,15.718,152.013
C04346=1098.939,97.710,439.902,176.698,15.718,152.014
C04347=1098.933,97.461,439.921,176.695,15.717,152.014
C04348=1098.927,97.212,439.938,176.692,15.717,152.015
C04349=1098.922,96.962,439.957,176.689,15.716,152.015
C04350=1098.916,96.714,439.975,176.687,15.717,152.016
C04351=1098.910,96.464,439.993,176.684,15.716,152.016
C04352=1098.904,96.190,440.013,176.681,15.715,152.017
C04353=1098.898,95.917,440.033,176.678,15.715,152.017
C04354=1098.891,95.643,440.052,176.675,15.715,152.018
C04355=1098.885,95.369,440.072,176.672,15.714,152.018
C04356=1098.879,95.119,440.090,176.670,15.714,152.019
C04357=1098.874,94.871,440.108,176.667,15.713,152.019
C04358=1098.869,94.621,440.126,176.664,15.714,152.020
C04359=1098.863,94.372,440.144,176.661,15.713,152.020
C04360=1098.857,94.123,440.162,176.659,15.713,152.021
C04361=1098.851,93.873,440.180,176.656,15.712,152.021
C04362=1098.846,93.623,440.198,176.653,15.712,152.022
C04363=1098.840,93.375,440.216,176.650,15.711,152.022
C04364=1098.834,93.125,440.234,176.648,15.711,152.023
C04365=1098.829,92.876,440.252,176.645,15.711,152.023
C04366=1098.823,92.626,440.270,176.643,15.710,152.024
C04367=1098.818,92.377,440.288,176.639,15.710,152.024
C04368=1098.812,92.128,440.305,176.637,15.710,152.025
C04369=1098.806,91.878,440.323,176.634,15.709,152.025
C04370=1098.801,91.629,440.341,176.632,15.709,152.026
C04371=1098.796,91.380,440.359,176.629,15.708,152.026
C04372=1098.789,91.131,440.378,176.627,15.708,152.027
C04373=1098.784,90.882,440.395,176.623,15.707,152.027
C04374=1098.778,90.632,440.413,176.621,15.707,152.028
C04375=1098.772,90.383,440.431,176.618,15.706,152.028
C04376=1098.767,90.134,440.448,176.616,15.706,152.029
C04377=1098.761,89.884,440.466,176.613,15.706,152.029
C04378=1098.755,89.635,440.484,176.610,15.706,152.030
C04379=1098.750,89.386,440.502,176.607,15.705,152.030
C04380=1098.744,89.136,440.519,176.605,15.705,152.031
C04381=1098.738,88.887,440.537,176.602,15.704,152.031
C04382=1098.732,88.638,440.555,176.600,15.704,152.032
C04383=1098.726,88.389,440.573,176.597,15.703,152.032
C04384=1098.721,88.140,440.590,176.594,15.703,152.033
C04385=1098.715,87.890,440.608,176.591,15.702,152.033
C04386=1098.709,87.641,440.626,176.589,15.702,152.033
C04387=1098.704,87.392,440.643,176.586,15.702,152.034
C04388=1098.698,87.142,440.661,176.583,15.701,152.034
C04389=1098.692,86.892,440.678,176.581,15.701,152.035
C04390=1098.687,86.643,440.695,176.578,15.701,152.035
C04391=1098.681,86.394,440.713,176.575,15.700,152.036
C04392=1098.675,86.145,440.731,176.573,15.700,152.036
C04393=1098.670,85.895,440.749,176.571,15.699,152.037
C04394=1098.664,85.646,440.766,176.567,15.699,152.037
C04395=1098.658,85.397,440.784,176.565,15.699,152.038
C04396=1098.653,85.148,440.802,176.562,15.698,152.038
C04397=1098.647,84.899,440.819,176.560,15.697,152.038
C04398=1098.641,84.648,440.836,176.557,15.697,152.039
C04399=1098.636,84.399,440.854,176.555,15.697,152.039
C04400=1098.630,84.150,440.872,176.552,15.696,152.040
C04401=1098.625,83.901,440.889,176.549,15.696,152.040
C04402=1098.619,83.651,440.907,176.546,15.695,152.041
C04403=1098.613,83.402,440.924,176.544,15.695,152.041
C04404=1098.608,83.153,440.941,176.541,15.694,152.042
C04405=1098.602,82.904,440.959,176.539,15.694,152.042
C04406=1098.595,82.654,440.976,176.536,15.693,152.043
C04407=1098.590,82.405,440.993,176.534,15.693,152.043
C04408=1098.585,82.156,441.011,176.531,15.692,152.043
C04409=1098.579,81.906,441.028,176.529,15.692,152.044
C04410=1098.574,81.657,441.046,176.526,15.691,152.044
C04411=1098.568,81.407,441.063,176.523,15.691,152.045
C04412=1098.562,81.158,441.081,176.521,15.691,152.045
C04413=1098.557,80.909,441.098,176.518,15.690,152.046
C04414=1098.552,80.659,441.115,176.516,15.689,152.046
C04415=1098.546,80.410,441.133,176.513,15.689,152.046
C04416=1098.539,80.136,441.152,176.510,15.688,152.047
C04417=1098.533,79.863,441.171,176.508,15.687,152.047
C04418=1098.527,79.589,441.189,176.504,15.687,152.048
C04419=1098.520,79.315,441.209,176.501,15.686,152.048
C04420=1098.515,79.066,441.226,176.499,15.686,152.049
C04421=1098.510,78.816,441.243,176.496,15.685,152.049
C04422=1098.504,78.567,441.261,176.494,15.685,152.050
C04423=1098.499,78.318,441.278,176.491,15.684,152.050
C04424=1098.493,78.069,441.295,176.489,15.684,152.050
C04425=1098.486,77.819,441.312,176.487,15.683,152.051
C04426=1098.481,77.569,441.329,176.484,15.682,152.051
C04427=1098.476,77.320,441.347,176.482,15.682,152.052
C04428=1098.470,77.071,441.363,176.479,15.681,152.052
C04429=1098.464,76.822,441.381,176.476,15.681,152.053
C04430=1098.458,76.572,441.398,176.473,15.681,152.053
C04431=1098.452,76.323,441.415,176.471,15.680,152.054
C04432=1098.447,76.073,441.432,176.468,15.680,152.054
C04433=1098.441,75.824,441.449,176.466,15.679,152.054
C04434=1098.435,75.575,441.466,176.463,15.678,152.055
C04435=1098.430,75.326,441.483,176.461,15.678,152.055
C04436=1098.425,75.076,441.500,176.458,15.678,152.056
C04437=1098.418,74.827,441.517,176.455,15.677,152.056
C04438=1098.413,74.577,441.534,176.453,15.677,152.056
C04439=1098.407,74.328,441.552,176.450,15.676,152.057
C04440=1098.401,74.079,441.568,176.448,15.675,152.057
C04441=1098.396,73.830,441.586,176.445,15.674,152.058
C04442=1098.390,73.580,441.602,176.443,15.674,152.058
C04443=1098.384,73.331,441.619,176.440,15.673,152.058
C04444=1098.379,73.082,441.636,176.438,15.673,152.059
C04445=1098.373,72.831,441.653,176.436,15.673,152.059
C04446=1098.367,72.582,441.670,176.433,15.672,152.060
C04447=1098.362,72.333,441.687,176.431,15.671,152.060
C04448=1098.355,72.084,441.704,176.428,15.671,152.061
C04449=1098.350,71.834,441.721,176.426,15.670,152.061
C04450=1098.345,71.585,441.738,176.423,15.669,152.061
C04451=1098.339,71.336,441.755,176.420,15.669,152.062
C04452=1098.334,71.086,441.772,176.418,15.668,152.062
C04453=1098.328,70.837,441.788,176.416,15.668,152.062
C04454=1098.322,70.588,441.806,176.413,15.667,152.063
C04455=1098.317,70.338,441.822,176.410,15.666,152.063
C04456=1098.311,70.089,441.839,176.408,15.666,152.064
C04457=1098.305,69.840,441.856,176.405,15.665,152.064
C04458=1098.299,69.591,441.873,176.403,15.665,152.065
C04459=1098.294,69.341,441.889,176.400,15.664,152.065
C04460=1098.288,69.091,441.906,176.398,15.663,152.065
C04461=1098.282,68.842,441.924,176.396,15.663,152.066
C04462=1098.276,68.592,441.940,176.393,15.662,152.066
C04463=1098.271,68.343,441.957,176.391,15.662,152.067
C04464=1098.265,68.093,441.973,176.388,15.661,152.067
C04465=1098.260,67.844,441.990,176.386,15.660,152.067
C04466=1098.254,67.595,442.007,176.383,15.660,152.068
C04467=1098.248,67.345,442.024,176.381,15.659,152.068
C04468=1098.242,67.096,442.040,176.378,15.658,152.069
C04469=1098.236,66.847,442.057,176.376,15.658,152.069
C04470=1098.231,66.598,442.074,176.374,15.658,152.069
C04471=1098.225,66.348,442.090,176.371,15.657,152.070
C04472=1098.220,66.099,442.107,176.369,15.656,152.070
C04473=1098.214,65.849,442.123,176.366,15.655,152.070
C04474=1098.209,65.600,442.140,176.364,15.655,152.071
C04475=1098.202,65.351,442.157,176.362,15.654,152.071
C04476=1098.196,65.102,442.173,176.359,15.654,152.072
C04477=1098.191,64.852,442.190,176.357,15.653,152.072
C04478=1098.185,64.603,442.206,176.354,15.652,152.072
C04479=1098.179,64.353,442.222,176.352,15.652,152.073
C04480=1098.174,64.079,442.241,176.349,15.651,152.073
C04481=1098.167,63.805,442.259,176.347,15.651,152.073
C04482=1098.161,63.531,442.277,176.344,15.650,152.074
C04483=1098.155,63.258,442.295,176.341,15.649,152.074
C04484=1098.149,63.008,442.311,176.338,15.649,152.075
C04485=1098.143,62.760,442.328,176.335,15.648,152.075
C04486=1098.137,62.510,442.345,176.333,15.648,152.076
C04487=1098.131,62.261,442.361,176.331,15.647,152.076
C04488=1098.126,62.011,442.378,176.328,15.646,152.076
C04489=1098.120,61.762,442.394,176.326,15.646,152.077
C04490=1098.114,61.513,442.410,176.323,15.645,152.077
C04491=1098.108,61.263,442.426,176.321,15.644,152.077
C04492=1098.102,61.014,442.443,176.319,15.644,152.078
C04493=1098.097,60.764,442.460,176.316,15.643,152.078
C04494=1098.091,60.515,442.476,176.314,15.643,152.079
C04495=1098.085,60.266,442.492,176.311,15.641,152.079
C04496=1098.079,60.016,442.508,176.309,15.641,152.079
C04497=1098.073,59.767,442.525,176.307,15.641,152.080
C04498=1098.067,59.517,442.541,176.304,15.640,152.080
C04499=1098.062,59.267,442.557,176.302,15.639,152.080
C04500=1098.056,59.018,442.573,176.299,15.638,152.081
C04501=1098.050,58.768,442.589,176.297,15.638,152.081
C04502=1098.044,58.519,442.606,176.295,15.637,152.082
C04503=1098.039,58.269,442.623,176.292,15.637,152.082
C04504=1098.033,58.020,442.639,176.290,15.636,152.082
C04505=1098.027,57.771,442.655,176.287,15.635,152.083
C04506=1098.021,57.521,442.671,176.285,15.634,152.083
C04507=1098.016,57.273,442.687,176.283,15.634,152.083
C04508=1098.010,57.023,442.703,176.280,15.633,152.084
C04509=1098.005,56.773,442.720,176.278,15.632,152.084
C04510=1097.999,56.524,442.736,176.275,15.632,152.084
C04511=1097.993,56.274,442.752,176.273,15.631,152.085
C04512=1097.987,56.025,442.768,176.271,15.631,152.085
C04513=1097.981,55.776,442.785,176.268,15.630,152.086
C04514=1097.975,55.526,442.800,176.266,15.629,152.086
C04515=1097.970,55.277,442.816,176.263,15.628,152.086
C04516=1097.964,55.028,442.832,176.262,15.627,152.087
C04517=1097.959,54.778,442.849,176.259,15.627,152.087
C04518=1097.953,54.529,442.865,176.257,15.626,152.087
C04519=1097.947,54.279,442.881,176.255,15.626,152.088
C04520=1097.941,54.029,442.897,176.253,15.625,152.088
C04521=1097.936,53.781,442.913,176.250,15.624,152.088
C04522=1097.930,53.531,442.929,176.248,15.623,152.089
C04523=1097.924,53.282,442.945,176.245,15.622,152.089
C04524=1097.918,53.032,442.961,176.243,15.622,152.089
C04525=1097.912,52.783,442.977,176.241,15.621,152.090
C04526=1097.907,52.533,442.993,176.238,15.620,152.090
C04527=1097.901,52.284,443.009,176.236,15.620,152.090
C04528=1097.895,52.035,443.025,176.233,15.618,152.091
C04529=1097.891,51.785,443.041,176.231,15.618,152.091
C04530=1097.885,51.535,443.058,176.229,15.617,152.091
C04531=1097.879,51.286,443.074,176.226,15.617,152.092
C04532=1097.874,51.037,443.089,176.224,15.616,152.092
C04533=1097.868,50.787,443.105,176.222,15.616,152.092
C04534=1097.862,50.538,443.121,176.219,15.614,152.093
C04535=1097.856,50.288,443.137,176.217,15.614,152.093
C04536=1097.851,50.039,443.153,176.215,15.613,152.093
C04537=1097.845,49.790,443.169,176.213,15.612,152.094
C04538=1097.839,49.540,443.185,176.211,15.612,152.094
C04539=1097.833,49.291,443.201,176.208,15.610,152.094
C04540=1097.828,49.041,443.216,176.206,15.610,152.095
C04541=1097.822,48.792,443.232,176.204,15.609,152.095
C04542=1097.816,48.542,443.248,176.201,15.608,152.095
C04543=1097.811,48.293,443.264,176.199,15.608,152.096
C04544=1097.804,48.019,443.281,176.196,15.607,152.096
C04545=1097.799,47.745,443.299,176.194,15.606,152.096
C04546=1097.792,47.471,443.316,176.191,15.605,152.097
C04547=1097.786,47.197,443.333,176.188,15.604,152.097
C04548=1097.780,46.947,443.349,176.187,15.603,152.097
C04549=1097.775,46.697,443.365,176.185,15.603,152.098
C04550=1097.769,46.449,443.381,176.182,15.602,152.098
C04551=1097.764,46.199,443.396,176.180,15.601,152.098
C04552=1097.758,45.949,443.413,176.178,15.600,152.099
C04553=1097.753,45.700,443.428,176.175,15.600,152.099
C04554=1097.747,45.451,443.444,176.173,15.599,152.099
C04555=1097.741,45.201,443.459,176.170,15.597,152.100
C04556=1097.736,44.952,443.475,176.169,15.597,152.100
C04557=1097.730,44.702,443.491,176.166,15.596,152.100
C04558=1097.724,44.452,443.506,176.164,15.595,152.100
C04559=1097.719,44.204,443.522,176.162,15.594,152.101
C04560=1097.713,43.954,443.538,176.160,15.594,152.101
C04561=1097.708,43.705,443.554,176.157,15.593,152.101
C04562=1097.702,43.455,443.569,176.155,15.592,152.102
C04563=1097.696,43.205,443.584,176.153,15.591,152.102
C04564=1097.690,42.956,443.601,176.150,15.591,152.102
C04565=1097.685,42.707,443.616,176.148,15.590,152.103
C04566=1097.679,42.457,443.631,176.146,15.588,152.103
C04567=1097.673,42.208,443.647,176.143,15.588,152.103
C04568=1097.668,41.958,443.662,176.142,15.588,152.104
C04569=1097.662,41.708,443.678,176.139,15.586,152.104
C04570=1097.656,41.459,443.694,176.137,15.586,152.104
C04571=1097.650,41.210,443.708,176.135,15.585,152.104
C04572=1097.645,40.960,443.724,176.132,15.584,152.105
C04573=1097.639,40.712,443.740,176.130,15.583,152.105
C04574=1097.634,40.462,443.755,176.128,15.583,152.105
C04575=1097.627,40.212,443.770,176.125,15.582,152.106
C04576=1097.622,39.963,443.786,176.124,15.581,152.106
C04577=1097.616,39.713,443.802,176.122,15.580,152.106
C04578=1097.611,39.463,443.817,176.119,15.579,152.107
C04579=1097.605,39.214,443.832,176.117,15.579,152.107
C04580=1097.599,38.965,443.848,176.115,15.578,152.107
C04581=1097.594,38.716,443.863,176.112,15.577,152.107
C04582=1097.588,38.466,443.879,176.110,15.576,152.108
C04583=1097.582,38.216,443.894,176.108,15.576,152.108
C04584=1097.577,37.967,443.909,176.106,15.574,152.108
C04585=1097.571,37.717,443.925,176.104,15.574,152.109
C04586=1097.565,37.469,443.940,176.102,15.573,152.109
C04587=1097.559,37.219,443.955,176.099,15.572,152.109
C04588=1097.553,36.969,443.970,176.097,15.571,152.110
C04589=1097.548,36.720,443.986,176.095,15.570,152.110
C04590=1097.542,36.470,444.002,176.092,15.569,152.110
C04591=1097.536,36.221,444.017,176.090,15.569,152.111
C04592=1097.530,35.971,444.032,176.088,15.568,152.111
C04593=1097.524,35.722,444.047,176.086,15.567,152.111
C04594=1097.519,35.472,444.062,176.084,15.566,152.111
C04595=1097.513,35.223,444.077,176.082,15.565,152.112
C04596=1097.508,34.974,444.092,176.079,15.565,152.112
C04597=1097.502,34.724,444.108,176.077,15.564,152.112
C04598=1097.495,34.475,444.123,176.075,15.563,152.113
C04599=1097.490,34.225,444.138,176.072,15.562,152.113
C04600=1097.484,33.976,444.153,176.071,15.561,152.113
C04601=1097.479,33.726,444.169,176.068,15.561,152.113
C04602=1097.472,33.477,444.184,176.066,15.560,152.114
C04603=1097.467,33.227,444.199,176.064,15.559,152.114
C04604=1097.461,32.978,444.214,176.062,15.558,152.114
C04605=1097.455,32.728,444.229,176.060,15.557,152.115
C04606=1097.450,32.479,444.244,176.057,15.556,152.115
C04607=1097.444,32.229,444.259,176.055,15.555,152.115
C04608=1097.438,31.955,444.276,176.052,15.554,152.116
C04609=1097.432,31.681,444.293,176.051,15.554,152.116
C04610=1097.425,31.408,444.309,176.048,15.552,152.116
C04611=1097.419,31.133,444.325,176.046,15.552,152.116
C04612=1097.413,30.883,444.340,176.043,15.550,152.117
C04613=1097.408,30.634,444.355,176.041,15.550,152.117
C04614=1097.401,30.384,444.370,176.039,15.549,152.117
C04615=1097.396,30.135,444.385,176.037,15.548,152.118
C04616=1097.390,29.885,444.400,176.035,15.547,152.118
C04617=1097.385,29.636,444.416,176.033,15.547,152.118
C04618=1097.379,29.386,444.431,176.031,15.546,152.118
C04619=1097.374,29.137,444.446,176.028,15.545,152.119
C04620=1097.367,28.888,444.461,176.026,15.544,152.119
C04621=1097.362,28.638,444.476,176.025,15.543,152.119
C04622=1097.356,28.389,444.491,176.022,15.542,152.119
C04623=1097.351,28.139,444.506,176.020,15.541,152.120
C04624=1097.345,27.889,444.520,176.018,15.540,152.120
C04625=1097.339,27.640,444.535,176.015,15.540,152.120
C04626=1097.333,27.390,444.550,176.013,15.539,152.121
C04627=1097.327,27.141,444.565,176.011,15.538,152.121
C04628=1097.321,26.892,444.580,176.009,15.537,152.121
C04629=1097.316,26.642,444.595,176.007,15.536,152.121
C04630=1097.310,26.393,444.610,176.005,15.535,152.122
C04631=1097.304,26.143,444.624,176.003,15.535,152.122
C04632=1097.299,25.894,444.639,176.000,15.533,152.122
C04633=1097.293,25.644,444.654,175.999,15.533,152.122
C04634=1097.287,25.395,444.669,175.997,15.532,152.123
C04635=1097.281,25.145,444.684,175.995,15.531,152.123
C04636=1097.276,24.896,444.698,175.992,15.530,152.123
C04637=1097.269,24.646,444.713,175.990,15.529,152.123
C04638=1097.264,24.397,444.728,175.988,15.528,152.124
C04639=1097.258,24.147,444.743,175.986,15.527,152.124
C04640=1097.253,23.897,444.757,175.984,15.526,152.124
C04641=1097.247,23.648,444.771,175.982,15.526,152.125
C04642=1097.241,23.399,444.787,175.980,15.525,152.125
C04643=1097.235,23.150,444.802,175.977,15.524,152.125
C04644=1097.229,22.899,444.816,175.975,15.523,152.125
C04645=1097.224,22.650,444.831,175.974,15.522,152.126
C04646=1097.218,22.401,444.846,175.971,15.521,152.126
C04647=1097.212,22.151,444.860,175.969,15.520,152.126
C04648=1097.207,21.902,444.874,175.967,15.519,152.126
C04649=1097.201,21.652,444.890,175.965,15.519,152.127
C04650=1097.195,21.403,444.904,175.963,15.517,152.127
C04651=1097.190,21.153,444.918,175.961,15.517,152.127
C04652=1097.183,20.904,444.933,175.959,15.516,152.127
C04653=1097.178,20.654,444.948,175.957,15.515,152.128
C04654=1097.172,20.404,444.963,175.954,15.514,152.128
C04655=1097.166,20.155,444.977,175.952,15.513,152.128
C04656=1097.161,19.906,444.991,175.950,15.512,152.128
C04657=1097.155,19.656,445.006,175.948,15.511,152.129
C04658=1097.149,19.407,445.021,175.946,15.510,152.129
C04659=1097.144,19.157,445.035,175.944,15.510,152.129
C04660=1097.138,18.907,445.050,175.942,15.509,152.130
C04661=1097.132,18.658,445.064,175.939,15.508,152.130
C04662=1097.126,18.408,445.079,175.938,15.507,152.130
C04663=1097.120,18.159,445.093,175.936,15.506,152.130
C04664=1097.115,17.910,445.107,175.934,15.505,152.131
C04665=1097.108,17.660,445.122,175.931,15.504,152.131
C04666=1097.103,17.410,445.137,175.929,15.503,152.131
C04667=1097.098,17.161,445.151,175.927,15.503,152.131
C04668=1097.092,16.911,445.166,175.925,15.502,152.132
C04669=1097.086,16.662,445.180,175.923,15.500,152.132
C04670=1097.080,16.412,445.194,175.921,15.499,152.132
C04671=1097.074,16.163,445.209,175.919,15.499,152.132
C04672=1097.068,15.890,445.224,175.917,15.497,152.133
C04673=1097.062,15.617,445.240,175.915,15.497,152.133
C04674=1097.056,15.345,445.256,175.912,15.495,152.133
C04675=1097.049,15.072,445.271,175.910,15.495,152.133
C04676=1097.043,14.823,445.286,175.908,15.494,152.134
C04677=1097.038,14.573,445.301,175.906,15.493,152.134
C04678=1097.032,14.324,445.315,175.904,15.492,152.134
C04679=1097.027,14.074,445.329,175.902,15.491,152.134
C04680=1097.019,13.825,445.343,175.900,15.491,152.135
C04681=1097.014,13.575,445.357,175.898,15.490,152.135
C04682=1097.008,13.326,445.371,175.895,15.488,152.135
C04683=1097.002,13.076,445.386,175.894,15.488,152.135
C04684=1096.997,12.826,445.400,175.892,15.487,152.136
C04685=1096.991,12.577,445.415,175.890,15.486,152.136
C04686=1096.985,12.327,445.429,175.887,15.485,152.136
C04687=1096.979,12.078,445.443,175.886,15.484,152.136
C04688=1096.974,11.829,445.457,175.884,15.483,152.137
C04689=1096.968,11.579,445.471,175.882,15.482,152.137
C04690=1096.962,11.329,445.486,175.879,15.481,152.137
C04691=1096.956,11.080,445.500,175.877,15.480,152.137
C04692=1096.951,10.830,445.514,175.875,15.480,152.138
C04693=1096.944,10.581,445.528,175.873,15.479,152.138
C04694=1096.938,10.331,445.542,175.871,15.478,152.138
C04695=1096.933,10.082,445.556,175.869,15.477,152.138
C04696=1096.926,9.832,445.571,175.867,15.476,152.139
C04697=1096.921,9.582,445.585,175.865,15.475,152.139
C04698=1096.915,9.333,445.599,175.864,15.474,152.139
C04699=1096.910,9.083,445.612,175.861,15.473,152.139
C04700=1096.903,8.834,445.627,175.859,15.472,152.140
C04701=1096.897,8.584,445.641,175.857,15.472,152.140
C04702=1096.892,8.335,445.655,175.855,15.471,152.140
C04703=1096.886,8.086,445.669,175.853,15.469,152.140
C04704=1096.880,7.836,445.683,175.851,15.468,152.141
C04705=1096.874,7.586,445.697,175.849,15.468,152.141
C04706=1096.869,7.336,445.711,175.847,15.467,152.141
C04707=1096.863,7.088,445.726,175.845,15.466,152.141
C04708=1096.857,6.838,445.739,175.843,15.465,152.142
C04709=1096.851,6.588,445.753,175.841,15.464,152.142
C04710=1096.845,6.338,445.767,175.839,15.463,152.142
C04711=1096.840,6.089,445.781,175.837,15.462,152.142
C04712=1096.834,5.840,445.795,175.835,15.461,152.142
C04713=1096.829,5.590,445.809,175.833,15.460,152.143
C04714=1096.822,5.340,445.823,175.831,15.459,152.143
C04715=1096.816,5.091,445.837,175.829,15.458,152.143
C04716=1096.811,4.841,445.851,175.827,15.458,152.143
C04717=1096.805,4.592,445.865,175.825,15.456,152.144
C04718=1096.800,4.342,445.878,175.823,15.455,152.144
C04719=1096.793,4.093,445.893,175.821,15.455,152.144
C04720=1096.787,3.843,445.907,175.819,15.454,152.144
C04721=1096.782,3.594,445.920,175.818,15.453,152.144
C04722=1096.776,3.344,445.934,175.815,15.452,152.145
C04723=1096.771,3.094,445.948,175.813,15.451,152.145
C04724=1096.765,2.845,445.961,175.811,15.450,152.145
C04725=1096.759,2.596,445.975,175.810,15.449,152.145
C04726=1096.753,2.345,445.990,175.808,15.448,152.146
C04727=1096.748,2.096,446.003,175.805,15.447,152.146
C04728=1096.742,1.846,446.017,175.803,15.446,152.146
C04729=1096.736,1.597,446.031,175.802,15.445,152.146
C04730=1096.730,1.348,446.045,175.800,15.444,152.147
C04731=1096.725,1.098,446.059,175.798,15.444,152.147
C04732=1096.719,0.849,446.073,175.795,15.442,152.147
C04733=1096.713,0.599,446.086,175.793,15.441,152.147
C04734=1096.707,0.349,446.100,175.792,15.440,152.147
C04735=1096.701,0.100,446.114,175.790,15.440,152.148
C04736=1096.696,-0.171,446.128,175.787,15.438,152.148
C04737=1096.689,-0.441,446.143,175.785,15.437,152.148
C04738=1096.683,-0.712,446.159,175.784,15.436,152.148
C04739=1096.677,-0.983,446.174,175.781,15.435,152.149
C04740=1096.671,-1.232,446.188,175.779,15.434,152.149
C04741=1096.665,-1.482,446.200,175.777,15.433,152.149
C04742=1096.660,-1.732,446.214,175.776,15.432,152.149
C04743=1096.655,-1.981,446.228,175.773,15.431,152.150
C04744=1096.648,-2.231,446.241,175.771,15.430,152.150
C04745=1096.643,-2.480,446.255,175.769,15.429,152.150
C04746=1096.637,-2.730,446.269,175.768,15.429,152.150
C04747=1096.632,-2.979,446.283,175.766,15.427,152.150
C04748=1096.626,-3.229,446.296,175.764,15.427,152.150
C04749=1096.620,-3.478,446.310,175.761,15.425,152.151
C04750=1096.613,-3.728,446.324,175.760,15.424,152.151
C04751=1096.608,-3.978,446.337,175.758,15.423,152.151
C04752=1096.602,-4.227,446.351,175.756,15.423,152.151
C04753=1096.597,-4.477,446.364,175.754,15.422,152.152
C04754=1096.590,-4.726,446.377,175.752,15.421,152.152
C04755=1096.585,-4.976,446.391,175.750,15.419,152.152
C04756=1096.579,-5.225,446.404,175.748,15.419,152.152
C04757=1096.573,-5.475,446.418,175.746,15.418,152.153
C04758=1096.567,-5.724,446.431,175.744,15.417,152.153
C04759=1096.561,-5.974,446.445,175.743,15.416,152.153
C04760=1096.555,-6.224,446.458,175.741,15.415,152.153
C04761=1096.549,-6.474,446.472,175.738,15.414,152.153
C04762=1096.543,-6.723,446.485,175.736,15.413,152.154
C04763=1096.538,-6.973,446.499,175.735,15.412,152.154
C04764=1096.532,-7.222,446.512,175.733,15.411,152.154
C04765=1096.526,-7.472,446.526,175.731,15.411,152.154
C04766=1096.520,-7.721,446.539,175.729,15.410,152.154
C04767=1096.515,-7.971,446.553,175.727,15.408,152.155
C04768=1096.508,-8.220,446.566,175.725,15.408,152.155
C04769=1096.503,-8.470,446.580,175.723,15.407,152.155
C04770=1096.497,-8.720,446.592,175.721,15.406,152.155
C04771=1096.492,-8.969,446.606,175.719,15.405,152.156
C04772=1096.485,-9.219,446.620,175.718,15.404,152.156
C04773=1096.480,-9.468,446.632,175.715,15.402,152.156
C04774=1096.474,-9.718,446.646,175.713,15.402,152.156
C04775=1096.468,-9.967,446.659,175.711,15.401,152.156
C04776=1096.462,-10.217,446.673,175.710,15.400,152.157
C04777=1096.456,-10.467,446.686,175.708,15.399,152.157
C04778=1096.451,-10.716,446.700,175.706,15.398,152.157
C04779=1096.445,-10.966,446.713,175.704,15.398,152.157
C04780=1096.439,-11.215,446.725,175.702,15.396,152.157
C04781=1096.433,-11.465,446.739,175.700,15.395,152.158
C04782=1096.427,-11.714,446.752,175.698,15.394,152.158
C04783=1096.422,-11.965,446.766,175.696,15.393,152.158
C04784=1096.416,-12.214,446.779,175.695,15.393,152.158
C04785=1096.410,-12.463,446.792,175.693,15.392,152.159
C04786=1096.404,-12.713,446.805,175.691,15.391,152.159
C04787=1096.398,-12.963,446.819,175.688,15.389,152.159
C04788=1096.393,-13.213,446.832,175.687,15.389,152.159
C04789=1096.387,-13.462,446.845,175.685,15.387,152.159
C04790=1096.381,-13.711,446.858,175.683,15.387,152.160
C04791=1096.375,-13.961,446.871,175.681,15.386,152.160
C04792=1096.370,-14.210,446.884,175.680,15.385,152.160
C04793=1096.365,-14.460,446.897,175.678,15.384,152.160
C04794=1096.358,-14.709,446.911,175.675,15.382,152.160
C04795=1096.352,-14.959,446.924,175.674,15.382,152.161
C04796=1096.347,-15.209,446.937,175.672,15.381,152.161
C04797=1096.341,-15.458,446.950,175.670,15.380,152.161
C04798=1096.335,-15.708,446.963,175.668,15.379,152.161
C04799=1096.329,-15.957,446.976,175.666,15.378,152.161
C04800=1096.322,-16.227,446.991,175.664,15.377,152.162
C04801=1096.317,-16.496,447.005,175.662,15.376,152.162
C04802=1096.310,-16.765,447.018,175.660,15.375,152.162
C04803=1096.303,-17.034,447.033,175.658,15.374,152.162
C04804=1096.298,-17.284,447.046,175.656,15.374,152.163
C04805=1096.291,-17.533,447.059,175.654,15.372,152.163
C04806=1096.285,-17.783,447.071,175.652,15.371,152.163
C04807=1096.280,-18.032,447.085,175.650,15.370,152.163
C04808=1096.275,-18.281,447.097,175.649,15.369,152.163
C04809=1096.269,-18.531,447.110,175.647,15.369,152.164
C04810=1096.263,-18.781,447.123,175.645,15.368,152.164
C04811=1096.257,-19.030,447.136,175.643,15.367,152.164
C04812=1096.251,-19.280,447.150,175.641,15.366,152.164
C04813=1096.245,-19.530,447.162,175.639,15.365,152.165
C04814=1096.239,-19.779,447.176,175.637,15.363,152.165
C04815=1096.233,-20.029,447.188,175.635,15.363,152.165
C04816=1096.227,-20.278,447.201,175.633,15.362,152.165
C04817=1096.221,-20.528,447.214,175.632,15.361,152.165
C04818=1096.216,-20.778,447.227,175.630,15.360,152.166
C04819=1096.210,-21.027,447.240,175.628,15.359,152.166
C04820=1096.204,-21.277,447.253,175.626,15.358,152.166
C04821=1096.198,-21.526,447.266,175.625,15.357,152.166
C04822=1096.192,-21.776,447.278,175.623,15.357,152.166
C04823=1096.186,-22.026,447.291,175.620,15.355,152.167
C04824=1096.180,-22.275,447.304,175.618,15.354,152.167
C04825=1096.175,-22.525,447.317,175.617,15.353,152.167
C04826=1096.170,-22.775,447.330,175.615,15.352,152.167
C04827=1096.163,-23.024,447.343,175.613,15.352,152.167
C04828=1096.157,-23.274,447.355,175.612,15.350,152.168
C04829=1096.152,-23.524,447.368,175.610,15.350,152.168
C04830=1096.145,-23.773,447.381,175.608,15.349,152.168
C04831=1096.140,-24.022,447.393,175.606,15.348,152.168
C04832=1096.134,-24.272,447.406,175.604,15.347,152.168
C04833=1096.129,-24.522,447.419,175.602,15.346,152.169
C04834=1096.123,-24.771,447.432,175.600,15.345,152.169
C04835=1096.117,-25.021,447.445,175.598,15.344,152.169
C04836=1096.111,-25.271,447.457,175.597,15.343,152.169
C04837=1096.105,-25.520,447.470,175.595,15.342,152.169
C04838=1096.099,-25.770,447.483,175.593,15.341,152.170
C04839=1096.093,-26.019,447.495,175.591,15.340,152.170
C04840=1096.088,-26.269,447.508,175.589,15.339,152.170
C04841=1096.082,-26.519,447.520,175.588,15.338,152.170
C04842=1096.076,-26.768,447.533,175.586,15.337,152.170
C04843=1096.070,-27.018,447.546,175.584,15.337,152.171
C04844=1096.064,-27.268,447.559,175.582,15.336,152.171
C04845=1096.058,-27.517,447.571,175.580,15.334,152.171
C04846=1096.052,-27.767,447.584,175.578,15.334,152.171
C04847=1096.047,-28.016,447.597,175.576,15.332,152.171
C04848=1096.041,-28.266,447.609,175.574,15.332,152.172
C04849=1096.035,-28.516,447.622,175.572,15.331,152.172
C04850=1096.029,-28.766,447.634,175.571,15.330,152.172
C04851=1096.023,-29.015,447.647,175.569,15.329,152.172
C04852=1096.018,-29.264,447.660,175.567,15.328,152.173
C04853=1096.012,-29.514,447.672,175.566,15.327,152.173
C04854=1096.006,-29.764,447.685,175.564,15.326,152.173
C04855=1096.000,-30.014,447.697,175.562,15.326,152.173
C04856=1095.993,-30.263,447.709,175.560,15.325,152.173
C04857=1095.988,-30.512,447.722,175.558,15.324,152.173
C04858=1095.982,-30.762,447.734,175.556,15.323,152.174
C04859=1095.976,-31.012,447.747,175.555,15.322,152.174
C04860=1095.970,-31.261,447.760,175.553,15.321,152.174
C04861=1095.965,-31.511,447.772,175.551,15.319,152.174
C04862=1095.959,-31.760,447.785,175.549,15.319,152.175
C04863=1095.953,-32.010,447.797,175.547,15.318,152.175
C04864=1095.946,-32.279,447.811,175.545,15.317,152.175
C04865=1095.940,-32.547,447.824,175.543,15.316,152.175
C04866=1095.934,-32.815,447.838,175.541,15.315,152.175
C04867=1095.927,-33.083,447.850,175.540,15.315,152.176
C04868=1095.921,-33.332,447.863,175.538,15.314,152.176
C04869=1095.915,-33.582,447.875,175.535,15.312,152.176
C04870=1095.910,-33.832,447.887,175.534,15.311,152.176
C04871=1095.904,-34.081,447.900,175.532,15.310,152.176
C04872=1095.898,-34.331,447.913,175.530,15.310,152.177
C04873=1095.892,-34.581,447.925,175.528,15.308,152.177
C04874=1095.886,-34.830,447.937,175.527,15.308,152.177
C04875=1095.880,-35.080,447.949,175.525,15.307,152.177
C04876=1095.874,-35.330,447.962,175.523,15.306,152.177
C04877=1095.869,-35.579,447.974,175.521,15.305,152.178
C04878=1095.863,-35.829,447.987,175.520,15.304,152.178
C04879=1095.857,-36.079,447.999,175.518,15.303,152.178
C04880=1095.851,-36.328,448.011,175.516,15.302,152.178
C04881=1095.845,-36.578,448.023,175.514,15.301,152.178
C04882=1095.839,-36.827,448.036,175.512,15.301,152.179
C04883=1095.834,-37.077,448.048,175.511,15.299,152.179
C04884=1095.828,-37.326,448.061,175.509,15.299,152.179
C04885=1095.822,-37.577,448.072,175.507,15.298,152.179
C04886=1095.816,-37.826,448.084,175.505,15.297,152.179
C04887=1095.811,-38.076,448.096,175.504,15.296,152.180
C04888=1095.805,-38.326,448.109,175.502,15.295,152.180
C04889=1095.799,-38.575,448.121,175.500,15.294,152.180
C04890=1095.793,-38.824,448.133,175.498,15.293,152.180
C04891=1095.787,-39.074,448.146,175.497,15.292,152.180
C04892=1095.781,-39.323,448.158,175.495,15.292,152.181
C04893=1095.775,-39.573,448.170,175.493,15.291,152.181
C04894=1095.769,-39.824,448.182,175.491,15.290,152.181
C04895=1095.764,-40.073,448.194,175.489,15.289,152.181
C04896=1095.757,-40.322,448.206,175.487,15.288,152.181
C04897=1095.751,-40.572,448.218,175.486,15.287,152.182
C04898=1095.745,-40.822,448.231,175.484,15.286,152.182
C04899=1095.739,-41.071,448.243,175.482,15.286,152.182
C04900=1095.733,-41.321,448.255,175.481,15.284,152.182
C04901=1095.728,-41.570,448.266,175.479,15.284,152.182
C04902=1095.722,-41.820,448.279,175.477,15.283,152.183
C04903=1095.716,-42.070,448.291,175.475,15.282,152.183
C04904=1095.710,-42.319,448.303,175.473,15.281,152.183
C04905=1095.704,-42.569,448.315,175.471,15.280,152.183
C04906=1095.698,-42.819,448.327,175.470,15.279,152.183
C04907=1095.692,-43.068,448.339,175.468,15.279,152.184
C04908=1095.686,-43.318,448.351,175.466,15.278,152.184
C04909=1095.680,-43.568,448.363,175.464,15.277,152.184
C04910=1095.675,-43.817,448.375,175.463,15.276,152.184
C04911=1095.669,-44.067,448.387,175.461,15.275,152.185
C04912=1095.663,-44.316,448.399,175.459,15.274,152.185
C04913=1095.657,-44.566,448.411,175.457,15.273,152.185
C04914=1095.651,-44.816,448.423,175.456,15.272,152.185
C04915=1095.645,-45.065,448.435,175.454,15.271,152.185
C04916=1095.639,-45.315,448.447,175.452,15.271,152.186
C04917=1095.633,-45.564,448.459,175.450,15.270,152.186
C04918=1095.628,-45.815,448.471,175.448,15.269,152.186
C04919=1095.621,-46.064,448.483,175.447,15.268,152.186
C04920=1095.616,-46.313,448.495,175.445,15.267,152.186
C04921=1095.609,-46.564,448.506,175.443,15.266,152.187
C04922=1095.604,-46.813,448.518,175.441,15.266,152.187
C04923=1095.597,-47.062,448.530,175.440,15.264,152.187
C04924=1095.592,-47.313,448.542,175.438,15.264,152.187
C04925=1095.586,-47.562,448.554,175.436,15.262,152.187
C04926=1095.580,-47.812,448.566,175.434,15.262,152.188
C04927=1095.575,-48.061,448.578,175.432,15.261,152.188
C04928=1095.568,-48.330,448.591,175.431,15.260,152.188
C04929=1095.562,-48.598,448.603,175.429,15.259,152.188
C04930=1095.556,-48.867,448.616,175.427,15.258,152.188
C04931=1095.549,-49.136,448.628,175.425,15.257,152.189
C04932=1095.543,-49.385,448.641,175.423,15.256,152.189
C04933=1095.537,-49.635,448.653,175.421,15.255,152.189
C04934=1095.532,-49.884,448.664,175.419,15.254,152.189
C04935=1095.525,-50.134,448.676,175.418,15.254,152.189
C04936=1095.520,-50.384,448.687,175.416,15.253,152.190
C04937=1095.513,-50.633,448.699,175.415,15.252,152.190
C04938=1095.508,-50.883,448.711,175.413,15.251,152.190
C04939=1095.502,-51.133,448.723,175.411,15.251,152.190
C04940=1095.496,-51.382,448.734,175.409,15.249,152.190
C04941=1095.490,-51.632,448.746,175.407,15.249,152.191
C04942=1095.484,-51.882,448.758,175.406,15.248,152.191
C04943=1095.478,-52.131,448.769,175.404,15.247,152.191
C04944=1095.471,-52.381,448.781,175.402,15.246,152.191
C04945=1095.466,-52.631,448.793,175.400,15.245,152.192
C04946=1095.459,-52.880,448.804,175.398,15.245,152.192
C04947=1095.453,-53.130,448.816,175.396,15.244,152.192
C04948=1095.448,-53.380,448.828,175.395,15.243,152.192
C04949=1095.442,-53.630,448.839,175.393,15.242,152.192
C04950=1095.435,-53.879,448.851,175.391,15.241,152.193
C04951=1095.429,-54.129,448.862,175.389,15.241,152.193
C04952=1095.424,-54.378,448.874,175.388,15.240,152.193
C04953=1095.417,-54.628,448.885,175.387,15.239,152.193
C04954=1095.411,-54.877,448.897,175.385,15.239,152.194
C04955=1095.405,-55.127,448.908,175.383,15.238,152.194
C04956=1095.399,-55.377,448.921,175.381,15.237,152.194
C04957=1095.393,-55.627,448.932,175.379,15.236,152.194
C04958=1095.387,-55.876,448.944,175.377,15.235,152.194
C04959=1095.381,-56.126,448.955,175.376,15.234,152.195
C04960=1095.375,-56.376,448.967,175.374,15.234,152.195
C04961=1095.369,-56.625,448.978,175.372,15.233,152.195
C04962=1095.363,-56.875,448.989,175.370,15.232,152.195
C04963=1095.357,-57.124,449.001,175.369,15.231,152.195
C04964=1095.351,-57.375,449.013,175.367,15.230,152.196
C04965=1095.345,-57.623,449.024,175.365,15.230,152.196
C04966=1095.339,-57.874,449.035,175.364,15.229,152.196
C04967=1095.333,-58.123,449.046,175.362,15.228,152.196
C04968=1095.327,-58.373,449.059,175.360,15.228,152.197
C04969=1095.322,-58.623,449.070,175.358,15.227,152.197
C04970=1095.315,-58.873,449.081,175.357,15.226,152.197
C04971=1095.309,-59.122,449.093,175.355,15.225,152.197
C04972=1095.304,-59.371,449.103,175.353,15.224,152.197
C04973=1095.298,-59.621,449.116,175.351,15.223,152.198
C04974=1095.292,-59.870,449.127,175.350,15.222,152.198
C04975=1095.286,-60.121,449.138,175.348,15.222,152.198
C04976=1095.279,-60.370,449.150,175.346,15.221,152.198
C04977=1095.273,-60.620,449.161,175.345,15.220,152.198
C04978=1095.268,-60.870,449.172,175.343,15.220,152.199
C04979=1095.262,-61.120,449.184,175.341,15.219,152.199
C04980=1095.256,-61.369,449.195,175.340,15.218,152.199
C04981=1095.249,-61.619,449.207,175.338,15.217,152.199
C04982=1095.244,-61.868,449.217,175.336,15.216,152.200
C04983=1095.238,-62.117,449.229,175.334,15.216,152.200
C04984=1095.232,-62.368,449.241,175.332,15.215,152.200
C04985=1095.226,-62.617,449.252,175.330,15.214,152.200
C04986=1095.220,-62.867,449.263,175.329,15.213,152.200
C04987=1095.214,-63.116,449.275,175.327,15.213,152.201
C04988=1095.208,-63.366,449.285,175.326,15.212,152.201
C04989=1095.202,-63.616,449.297,175.324,15.211,152.201
C04990=1095.196,-63.865,449.308,175.322,15.210,152.201
C04991=1095.190,-64.115,449.320,175.321,15.209,152.201
C04992=1095.184,-64.385,449.331,175.319,15.209,152.202
C04993=1095.178,-64.655,449.343,175.317,15.208,152.202
C04994=1095.171,-64.925,449.356,175.315,15.207,152.202
C04995=1095.164,-65.194,449.368,175.313,15.206,152.202
C04996=1095.159,-65.444,449.379,175.311,15.205,152.203
C04997=1095.153,-65.694,449.391,175.310,15.205,152.203
C04998=1095.147,-65.944,449.401,175.308,15.204,152.203
C04999=1095.141,-66.193,449.413,175.306,15.203,152.203
C05000=1095.135,-66.443,449.424,175.304,15.202,152.203
C05001=1095.129,-66.692,449.435,175.303,15.202,152.204
C05002=1095.123,-66.943,449.446,175.301,15.201,152.204
C05003=1095.117,-67.192,449.457,175.300,15.200,152.204
C05004=1095.111,-67.442,449.468,175.298,15.199,152.204
C05005=1095.106,-67.692,449.480,175.296,15.199,152.205
C05006=1095.100,-67.941,449.492,175.294,15.197,152.205
C05007=1095.094,-68.190,449.502,175.292,15.197,152.205
C05008=1095.088,-68.441,449.514,175.290,15.196,152.205
C05009=1095.082,-68.690,449.525,175.289,15.196,152.205
C05010=1095.076,-68.940,449.535,175.288,15.195,152.205
C05011=1095.070,-69.190,449.547,175.286,15.194,152.206
C05012=1095.064,-69.439,449.558,175.284,15.193,152.206
C05013=1095.058,-69.689,449.568,175.282,15.193,152.206
C05014=1095.053,-69.938,449.579,175.281,15.191,152.206
C05015=1095.046,-70.188,449.591,175.279,15.191,152.207
C05016=1095.040,-70.438,449.601,175.278,15.191,152.207
C05017=1095.035,-70.687,449.612,175.276,15.189,152.207
C05018=1095.029,-70.938,449.624,175.274,15.189,152.207
C05019=1095.023,-71.187,449.635,175.272,15.188,152.208
C05020=1095.018,-71.437,449.646,175.270,15.187,152.208
C05021=1095.012,-71.686,449.657,175.269,15.186,152.208
C05022=1095.006,-71.937,449.668,175.268,15.186,152.208
C05023=1095.000,-72.186,449.679,175.266,15.185,152.208
C05024=1094.994,-72.436,449.690,175.264,15.184,152.208
C05025=1094.988,-72.686,449.701,175.262,15.183,152.209
C05026=1094.982,-72.935,449.712,175.260,15.183,152.209
C05027=1094.976,-73.185,449.723,175.258,15.182,152.209
C05028=1094.971,-73.434,449.734,175.257,15.181,152.209
C05029=1094.965,-73.684,449.745,175.256,15.181,152.210
C05030=1094.958,-73.934,449.756,175.254,15.180,152.210
C05031=1094.953,-74.183,449.767,175.252,15.179,152.210
C05032=1094.947,-74.433,449.778,175.250,15.178,152.210
C05033=1094.941,-74.683,449.789,175.249,15.177,152.210
C05034=1094.935,-74.933,449.800,175.247,15.177,152.211
C05035=1094.928,-75.182,449.810,175.246,15.177,152.211
C05036=1094.923,-75.431,449.821,175.244,15.176,152.211
C05037=1094.916,-75.681,449.832,175.242,15.175,152.211
C05038=1094.911,-75.931,449.843,175.240,15.174,152.212
C05039=1094.905,-76.180,449.854,175.238,15.173,152.212
C05040=1094.899,-76.431,449.865,175.237,15.173,152.212
C05041=1094.893,-76.680,449.876,175.235,15.173,152.212
C05042=1094.886,-76.929,449.886,175.233,15.172,152.213
C05043=1094.881,-77.179,449.896,175.232,15.171,152.213
C05044=1094.875,-77.430,449.908,175.230,15.170,152.213
C05045=1094.869,-77.679,449.919,175.229,15.170,152.213
C05046=1094.863,-77.929,449.929,175.227,15.169,152.213
C05047=1094.857,-78.178,449.940,175.225,15.168,152.214
C05048=1094.850,-78.428,449.951,175.223,15.168,152.214
C05049=1094.845,-78.677,449.962,175.222,15.167,152.214
C05050=1094.839,-78.927,449.972,175.220,15.167,152.214
C05051=1094.833,-79.177,449.983,175.219,15.166,152.215
C05052=1094.827,-79.427,449.994,175.217,15.165,152.215
C05053=1094.821,-79.676,450.004,175.215,15.164,152.215
C05054=1094.815,-79.926,450.015,175.213,15.163,152.215
C05055=1094.809,-80.175,450.026,175.212,15.163,152.215
C05056=1094.803,-80.448,450.037,175.210,15.162,152.216
C05057=1094.796,-80.720,450.049,175.208,15.162,152.216
C05058=1094.789,-80.992,450.061,175.206,15.161,152.216
C05059=1094.782,-81.264,450.072,175.205,15.160,152.217
C05060=1094.776,-81.514,450.083,175.203,15.160,152.217
C05061=1094.770,-81.763,450.094,175.201,15.159,152.217
C05062=1094.763,-82.013,450.104,175.199,15.158,152.217
C05063=1094.758,-82.263,450.115,175.198,15.158,152.218
C05064=1094.752,-82.513,450.125,175.196,15.157,152.218
C05065=1094.746,-82.762,450.136,175.194,15.157,152.218
C05066=1094.739,-83.012,450.147,175.192,15.156,152.218
C05067=1094.734,-83.262,450.157,175.191,15.156,152.219
C05068=1094.727,-83.511,450.167,175.189,15.155,152.219
C05069=1094.722,-83.761,450.178,175.188,15.154,152.219
C05070=1094.715,-84.010,450.189,175.186,15.153,152.219
C05071=1094.709,-84.261,450.199,175.184,15.153,152.219
C05072=1094.703,-84.510,450.210,175.183,15.153,152.220
C05073=1094.697,-84.759,450.220,175.181,15.152,152.220
C05074=1094.692,-85.009,450.230,175.179,15.151,152.220
C05075=1094.685,-85.260,450.242,175.177,15.151,152.220
C05076=1094.679,-85.509,450.252,175.176,15.150,152.221
C05077=1094.673,-85.758,450.263,175.174,15.150,152.221
C05078=1094.667,-86.008,450.272,175.172,15.149,152.221
C05079=1094.661,-86.258,450.283,175.170,15.148,152.221
C05080=1094.655,-86.508,450.295,175.169,15.148,152.222
C05081=1094.649,-86.758,450.304,175.168,15.147,152.222
C05082=1094.643,-87.007,450.315,175.166,15.146,152.222
C05083=1094.637,-87.257,450.325,175.164,15.146,152.222
C05084=1094.631,-87.506,450.335,175.163,15.146,152.223
C05085=1094.624,-87.756,450.346,175.161,15.145,152.223
C05086=1094.618,-88.006,450.356,175.159,15.144,152.223
C05087=1094.613,-88.256,450.367,175.157,15.143,152.223
C05088=1094.606,-88.505,450.377,175.156,15.143,152.224
C05089=1094.601,-88.755,450.388,175.154,15.143,152.224
C05090=1094.594,-89.004,450.398,175.152,15.142,152.224
C05091=1094.589,-89.254,450.408,175.150,15.141,152.224
C05092=1094.582,-89.504,450.419,175.149,15.141,152.225
C05093=1094.576,-89.754,450.430,175.147,15.140,152.225
C05094=1094.571,-90.004,450.440,175.146,15.139,152.225
C05095=1094.564,-90.253,450.450,175.144,15.139,152.225
C05096=1094.559,-90.503,450.460,175.143,15.139,152.225
C05097=1094.552,-90.752,450.470,175.141,15.138,152.226
C05098=1094.547,-91.002,450.481,175.139,15.137,152.226
C05099=1094.540,-91.252,450.491,175.138,15.137,152.226
C05100=1094.534,-91.502,450.502,175.136,15.136,152.226
C05101=1094.528,-91.752,450.512,175.134,15.136,152.227
C05102=1094.522,-92.001,450.523,175.132,15.135,152.227
C05103=1094.516,-92.251,450.532,175.131,15.135,152.227
C05104=1094.510,-92.500,450.543,175.129,15.134,152.228
C05105=1094.504,-92.750,450.553,175.127,15.133,152.228
C05106=1094.498,-93.000,450.563,175.126,15.133,152.228
C05107=1094.492,-93.249,450.573,175.124,15.133,152.228
C05108=1094.486,-93.499,450.584,175.122,15.132,152.229
C05109=1094.480,-93.749,450.593,175.120,15.131,152.229
C05110=1094.474,-93.999,450.605,175.119,15.131,152.229
C05111=1094.468,-94.249,450.614,175.117,15.131,152.229
C05112=1094.462,-94.498,450.625,175.115,15.130,152.230
C05113=1094.456,-94.748,450.635,175.114,15.130,152.230
C05114=1094.450,-94.998,450.645,175.113,15.129,152.230
C05115=1094.444,-95.247,450.655,175.111,15.128,152.230
C05116=1094.438,-95.497,450.665,175.109,15.127,152.230
C05117=1094.432,-95.747,450.676,175.108,15.127,152.231
C05118=1094.426,-95.997,450.686,175.106,15.126,152.231
C05119=1094.420,-96.246,450.696,175.104,15.126,152.231
C05120=1094.414,-96.520,450.708,175.102,15.125,152.231
C05121=1094.407,-96.795,450.718,175.101,15.125,152.232
C05122=1094.401,-97.070,450.730,175.099,15.125,152.232
C05123=1094.394,-97.344,450.740,175.097,15.124,152.232
C05124=1094.388,-97.593,450.751,175.095,15.123,152.233
C05125=1094.382,-97.843,450.761,175.094,15.123,152.233
C05126=1094.376,-98.093,450.771,175.092,15.123,152.233
C05127=1094.370,-98.342,450.781,175.090,15.122,152.233
C05128=1094.364,-98.592,450.791,175.088,15.121,152.234
C05129=1094.357,-98.842,450.801,175.087,15.121,152.234
C05130=1094.351,-99.092,450.811,175.085,15.120,152.234
C05131=1094.346,-99.342,450.821,175.083,15.120,152.234
C05132=1094.339,-99.591,450.832,175.082,15.120,152.235
C05133=1094.333,-99.841,450.841,175.080,15.119,152.235
C05134=1094.327,-100.091,450.851,175.079,15.118,152.235
C05135=1094.321,-100.340,450.862,175.077,15.118,152.235
C05136=1094.315,-100.590,450.871,175.076,15.117,152.236
C05137=1094.309,-100.840,450.881,175.074,15.117,152.236
C05138=1094.303,-101.089,450.892,175.073,15.117,152.236
C05139=1094.297,-101.339,450.901,175.071,15.116,152.236
C05140=1094.291,-101.589,450.911,175.068,15.116,152.237
C05141=1094.285,-101.839,450.921,175.067,15.116,152.237
C05142=1094.279,-102.088,450.931,175.065,15.115,152.237
C05143=1094.272,-102.338,450.941,175.064,15.114,152.238
C05144=1094.266,-102.588,450.950,175.062,15.114,152.238
C05145=1094.261,-102.837,450.961,175.061,15.113,152.238
C05146=1094.254,-103.087,450.971,175.059,15.113,152.238
C05147=1094.248,-103.337,450.980,175.058,15.113,152.239
C05148=1094.243,-103.587,450.991,175.056,15.112,152.239
C05149=1094.236,-103.836,451.001,175.055,15.112,152.239
C05150=1094.230,-104.086,451.010,175.053,15.111,152.239
C05151=1094.224,-104.336,451.020,175.050,15.111,152.240
C05152=1094.218,-104.585,451.030,175.049,15.111,152.240
C05153=1094.212,-104.835,451.040,175.047,15.110,152.240
C05154=1094.206,-105.085,451.050,175.046,15.110,152.241
C05155=1094.200,-105.334,451.060,175.044,15.109,152.241
C05156=1094.194,-105.584,451.069,175.043,15.109,152.241
C05157=1094.188,-105.834,451.080,175.041,15.108,152.241
C05158=1094.182,-106.083,451.090,175.040,15.108,152.242
C05159=1094.175,-106.333,451.099,175.038,15.107,152.242
C05160=1094.169,-106.583,451.109,175.035,15.107,152.242
C05161=1094.163,-106.833,451.118,175.034,15.107,152.242
C05162=1094.158,-107.083,451.128,175.032,15.106,152.243
C05163=1094.151,-107.332,451.139,175.031,15.106,152.243
C05164=1094.145,-107.582,451.148,175.029,15.105,152.243
C05165=1094.139,-107.832,451.158,175.028,15.105,152.243
C05166=1094.133,-108.082,451.167,175.026,15.105,152.244
C05167=1094.127,-108.331,451.177,175.024,15.105,152.244
C05168=1094.120,-108.581,451.187,175.022,15.104,152.244
C05169=1094.115,-108.831,451.197,175.021,15.104,152.245
C05170=1094.108,-109.080,451.207,175.019,15.103,152.245
C05171=1094.102,-109.330,451.217,175.018,15.103,152.245
C05172=1094.096,-109.580,451.226,175.016,15.102,152.245
C05173=1094.090,-109.830,451.236,175.014,15.102,152.246
C05174=1094.084,-110.080,451.245,175.013,15.102,152.246
C05175=1094.078,-110.329,451.255,175.011,15.101,152.246
C05176=1094.071,-110.579,451.264,175.010,15.101,152.247
C05177=1094.065,-110.828,451.275,175.008,15.101,152.247
C05178=1094.059,-111.078,451.284,175.006,15.100,152.247
C05179=1094.053,-111.328,451.294,175.005,15.100,152.247
C05180=1094.046,-111.578,451.303,175.003,15.100,152.248
C05181=1094.041,-111.828,451.314,175.002,15.099,152.248
C05182=1094.035,-112.078,451.323,175.000,15.099,152.248
C05183=1094.029,-112.328,451.333,174.998,15.099,152.249
C05184=1094.022,-112.592,451.343,174.997,15.098,152.249
C05185=1094.016,-112.859,451.353,174.995,15.098,152.249
C05186=1094.009,-113.124,451.363,174.993,15.097,152.249
C05187=1094.002,-113.390,451.373,174.991,15.098,152.250
C05188=1093.996,-113.639,451.383,174.990,15.097,152.250
C05189=1093.990,-113.889,451.392,174.988,15.096,152.250
C05190=1093.984,-114.138,451.402,174.987,15.096,152.251
C05191=1093.978,-114.388,451.411,174.985,15.095,152.251
C05192=1093.972,-114.638,451.421,174.983,15.096,152.251
C05193=1093.966,-114.888,451.431,174.981,15.095,152.251
C05194=1093.959,-115.138,451.440,174.979,15.094,152.252
C05195=1093.953,-115.387,451.450,174.978,15.094,152.252
C05196=1093.947,-115.637,451.459,174.976,15.094,152.252
C05197=1093.941,-115.887,451.469,174.975,15.094,152.253
C05198=1093.935,-116.137,451.478,174.973,15.093,152.253
C05199=1093.928,-116.387,451.488,174.972,15.093,152.253
C05200=1093.923,-116.636,451.496,174.970,15.093,152.254
C05201=1093.917,-116.886,451.506,174.968,15.092,152.254
C05202=1093.911,-117.136,451.516,174.967,15.092,152.254
C05203=1093.905,-117.386,451.525,174.965,15.092,152.254
C05204=1093.899,-117.635,451.535,174.963,15.092,152.255
C05205=1093.892,-117.885,451.544,174.962,15.091,152.255
C05206=1093.886,-118.135,451.554,174.960,15.091,152.255
C05207=1093.880,-118.385,451.563,174.958,15.091,152.256
C05208=1093.874,-118.635,451.573,174.956,15.090,152.256
C05209=1093.868,-118.884,451.583,174.955,15.090,152.256
C05210=1093.862,-119.134,451.592,174.953,15.090,152.257
C05211=1093.855,-119.383,451.601,174.952,15.090,152.257
C05212=1093.849,-119.633,451.610,174.950,15.089,152.257
C05213=1093.843,-119.883,451.620,174.949,15.089,152.257
C05214=1093.837,-120.133,451.629,174.947,15.089,152.258
C05215=1093.831,-120.383,451.638,174.946,15.089,152.258
C05216=1093.825,-120.633,451.648,174.944,15.088,152.258
C05217=1093.818,-120.882,451.657,174.942,15.088,152.259
C05218=1093.813,-121.132,451.667,174.940,15.088,152.259
C05219=1093.807,-121.381,451.676,174.939,15.087,152.259
C05220=1093.800,-121.631,451.685,174.937,15.088,152.260
C05221=1093.794,-121.881,451.694,174.935,15.087,152.260
C05222=1093.788,-122.131,451.704,174.934,15.087,152.260
C05223=1093.782,-122.381,451.713,174.932,15.087,152.260
C05224=1093.775,-122.631,451.723,174.931,15.087,152.261
C05225=1093.770,-122.880,451.732,174.929,15.086,152.261
C05226=1093.763,-123.129,451.741,174.927,15.086,152.261
C05227=1093.757,-123.380,451.750,174.926,15.086,152.262
C05228=1093.751,-123.629,451.759,174.924,15.086,152.262
C05229=1093.745,-123.879,451.769,174.922,15.085,152.262
C05230=1093.739,-124.129,451.778,174.920,15.085,152.263
C05231=1093.733,-124.378,451.788,174.919,15.085,152.263
C05232=1093.726,-124.628,451.796,174.917,15.084,152.263
C05233=1093.720,-124.878,451.805,174.916,15.084,152.263
C05234=1093.714,-125.128,451.815,174.914,15.084,152.264
C05235=1093.708,-125.378,451.825,174.913,15.084,152.264
C05236=1093.702,-125.627,451.834,174.911,15.083,152.264
C05237=1093.695,-125.878,451.842,174.909,15.084,152.265
C05238=1093.690,-126.127,451.852,174.907,15.083,152.265
C05239=1093.683,-126.376,451.861,174.906,15.083,152.265
C05240=1093.676,-126.626,451.870,174.904,15.083,152.266
C05241=1093.671,-126.876,451.879,174.903,15.083,152.266
C05242=1093.664,-127.126,451.889,174.901,15.083,152.266
C05243=1093.659,-127.375,451.898,174.900,15.082,152.267
C05244=1093.652,-127.636,451.907,174.897,15.082,152.267
C05245=1093.645,-127.896,451.917,174.896,15.082,152.267
C05246=1093.639,-128.156,451.926,174.894,15.081,152.267
C05247=1093.642,-128.415,451.939,174.894,15.079,152.267
C05248=1093.235,-128.436,451.824,174.849,15.187,152.298
C05249=1093.232,-128.178,451.812,174.849,15.191,152.298
C05250=1093.238,-127.917,451.802,174.851,15.191,152.298
C05251=1093.244,-127.658,451.793,174.853,15.192,152.297
C05252=1093.250,-127.398,451.784,174.854,15.192,152.297
C05253=1093.256,-127.148,451.774,174.857,15.192,152.297
C05254=1093.263,-126.898,451.765,174.858,15.192,152.297
C05255=1093.269,-126.649,451.756,174.860,15.192,152.296
C05256=1093.275,-126.398,451.747,174.861,15.192,152.296
C05257=1093.281,-126.149,451.737,174.863,15.193,152.296
C05258=1093.288,-125.900,451.729,174.864,15.192,152.295
C05259=1093.294,-125.650,451.719,174.866,15.193,152.295
C05260=1093.300,-125.399,451.710,174.867,15.193,152.295
C05261=1093.306,-125.150,451.701,174.870,15.193,152.294
C05262=1093.313,-124.900,451.692,174.871,15.193,152.294
C05263=1093.319,-124.650,451.682,174.873,15.194,152.294
C05264=1093.324,-124.401,451.673,174.874,15.194,152.293
C05265=1093.330,-124.151,451.664,174.876,15.194,152.293
C05266=1093.337,-123.901,451.654,174.878,15.195,152.293
C05267=1093.344,-123.651,451.645,174.879,15.195,152.293
C05268=1093.350,-123.402,451.636,174.881,15.195,152.292
C05269=1093.356,-123.151,451.627,174.882,15.195,152.292
C05270=1093.361,-122.902,451.618,174.884,15.196,152.292
C05271=1093.367,-122.652,451.608,174.886,15.196,152.291
C05272=1093.373,-122.403,451.599,174.887,15.196,152.291
C05273=1093.380,-122.153,451.590,174.889,15.196,152.291
C05274=1093.387,-121.903,451.580,174.891,15.197,152.290
C05275=1093.392,-121.653,451.571,174.892,15.197,152.290
C05276=1093.398,-121.404,451.562,174.894,15.197,152.290
C05277=1093.404,-121.154,451.552,174.896,15.198,152.290
C05278=1093.410,-120.904,451.543,174.897,15.198,152.289
C05279=1093.416,-120.654,451.533,174.899,15.198,152.289
C05280=1093.423,-120.405,451.524,174.900,15.198,152.289
C05281=1093.430,-120.155,451.515,174.902,15.199,152.288
C05282=1093.435,-119.905,451.506,174.903,15.199,152.288
C05283=1093.442,-119.655,451.496,174.905,15.199,152.288
C05284=1093.447,-119.406,451.487,174.907,15.200,152.288
C05285=1093.453,-119.156,451.478,174.909,15.200,152.287
C05286=1093.460,-118.906,451.468,174.910,15.200,152.287
C05287=1093.466,-118.656,451.458,174.912,15.200,152.287
C05288=1093.472,-118.407,451.449,174.913,15.201,152.286
C05289=1093.478,-118.157,451.439,174.915,15.201,152.286
C05290=1093.484,-117.907,451.430,174.917,15.201,152.286
C05291=1093.490,-117.657,451.420,174.918,15.201,152.286
C05292=1093.497,-117.408,451.411,174.920,15.202,152.285
C05293=1093.503,-117.159,451.402,174.922,15.202,152.285
C05294=1093.509,-116.909,451.392,174.923,15.202,152.285
C05295=1093.515,-116.658,451.384,174.925,15.203,152.284
C05296=1093.521,-116.409,451.374,174.926,15.203,152.284
C05297=1093.527,-116.159,451.364,174.928,15.204,152.284
C05298=1093.533,-115.909,451.355,174.930,15.204,152.283
C05299=1093.540,-115.659,451.345,174.931,15.204,152.283
C05300=1093.546,-115.409,451.336,174.933,15.205,152.283
C05301=1093.552,-115.160,451.326,174.934,15.205,152.283
C05302=1093.558,-114.910,451.317,174.937,15.205,152.282
C05303=1093.564,-114.660,451.307,174.938,15.205,152.282
C05304=1093.570,-114.410,451.298,174.940,15.206,152.282
C05305=1093.576,-114.161,451.288,174.941,15.206,152.282
C05306=1093.582,-113.911,451.279,174.943,15.207,152.281
C05307=1093.588,-113.662,451.269,174.944,15.207,152.281
C05308=1093.595,-113.412,451.260,174.946,15.207,152.281
C05309=1093.601,-113.146,451.249,174.948,15.208,152.280
C05310=1093.607,-112.880,451.239,174.950,15.208,152.280
C05311=1093.614,-112.614,451.228,174.952,15.209,152.280
C05312=1093.621,-112.348,451.218,174.953,15.208,152.279
C05313=1093.627,-112.098,451.209,174.955,15.209,152.279
C05314=1093.633,-111.848,451.199,174.957,15.210,152.279
C05315=1093.639,-111.598,451.189,174.958,15.210,152.279
C05316=1093.645,-111.348,451.180,174.960,15.211,152.278
C05317=1093.651,-111.099,451.170,174.961,15.211,152.278
C05318=1093.657,-110.849,451.160,174.963,15.211,152.278
C05319=1093.663,-110.599,451.151,174.965,15.212,152.278
C05320=1093.670,-110.350,451.141,174.966,15.212,152.277
C05321=1093.676,-110.100,451.131,174.968,15.212,152.277
C05322=1093.682,-109.850,451.121,174.969,15.212,152.277
C05323=1093.688,-109.600,451.112,174.971,15.213,152.277
C05324=1093.694,-109.351,451.102,174.973,15.214,152.276
C05325=1093.701,-109.101,451.093,174.974,15.214,152.276
C05326=1093.707,-108.851,451.083,174.976,15.215,152.276
C05327=1093.712,-108.601,451.073,174.978,15.215,152.275
C05328=1093.719,-108.352,451.063,174.979,15.215,152.275
C05329=1093.725,-108.102,451.053,174.981,15.216,152.275
C05330=1093.731,-107.852,451.044,174.982,15.216,152.275
C05331=1093.737,-107.602,451.034,174.984,15.216,152.274
C05332=1093.743,-107.353,451.024,174.986,15.217,152.274
C05333=1093.749,-107.103,451.015,174.987,15.217,152.274
C05334=1093.755,-106.853,451.004,174.989,15.218,152.274
C05335=1093.761,-106.603,450.994,174.991,15.218,152.273
C05336=1093.768,-106.354,450.985,174.992,15.219,152.273
C05337=1093.774,-106.104,450.975,174.994,15.219,152.273
C05338=1093.780,-105.854,450.966,174.996,15.219,152.272
C05339=1093.785,-105.605,450.955,174.997,15.219,152.272
C05340=1093.791,-105.356,450.946,174.999,15.220,152.272
C05341=1093.797,-105.106,450.936,175.001,15.221,152.272
C05342=1093.804,-104.856,450.927,175.002,15.221,152.271
C05343=1093.809,-104.606,450.916,175.004,15.222,152.271
C05344=1093.815,-104.357,450.906,175.005,15.222,152.271
C05345=1093.822,-104.107,450.897,175.007,15.222,152.271
C05346=1093.828,-103.857,450.887,175.009,15.223,152.270
C05347=1093.834,-103.607,450.877,175.010,15.223,152.270
C05348=1093.840,-103.357,450.866,175.012,15.224,152.270
C05349=1093.847,-103.107,450.857,175.014,15.225,152.270
C05350=1093.853,-102.857,450.847,175.015,15.225,152.269
C05351=1093.858,-102.607,450.837,175.017,15.225,152.269
C05352=1093.865,-102.358,450.827,175.019,15.226,152.269
C05353=1093.871,-102.108,450.817,175.020,15.226,152.269
C05354=1093.877,-101.859,450.807,175.022,15.227,152.268
C05355=1093.883,-101.609,450.797,175.024,15.227,152.268
C05356=1093.889,-101.359,450.787,175.025,15.228,152.268
C05357=1093.895,-101.109,450.777,175.027,15.228,152.268
C05358=1093.901,-100.860,450.767,175.028,15.229,152.267
C05359=1093.907,-100.610,450.757,175.030,15.229,152.267
C05360=1093.913,-100.360,450.747,175.031,15.230,152.267
C05361=1093.920,-100.111,450.737,175.033,15.230,152.267
C05362=1093.925,-99.861,450.727,175.036,15.231,152.266
C05363=1093.931,-99.611,450.717,175.037,15.231,152.266
C05364=1093.938,-99.362,450.707,175.039,15.231,152.266
C05365=1093.943,-99.112,450.697,175.040,15.232,152.265
C05366=1093.949,-98.862,450.687,175.042,15.232,152.265
C05367=1093.956,-98.613,450.677,175.043,15.233,152.265
C05368=1093.962,-98.363,450.668,175.045,15.233,152.265
C05369=1093.968,-98.112,450.657,175.046,15.234,152.264
C05370=1093.974,-97.863,450.647,175.048,15.234,152.264
C05371=1093.981,-97.613,450.637,175.050,15.235,152.264
C05372=1093.986,-97.364,450.626,175.051,15.236,152.264
C05373=1093.993,-97.089,450.616,175.053,15.236,152.264
C05374=1093.999,-96.815,450.605,175.055,15.237,152.263
C05375=1094.006,-96.541,450.593,175.057,15.237,152.263
C05376=1094.012,-96.266,450.582,175.059,15.238,152.263
C05377=1094.018,-96.017,450.572,175.060,15.239,152.263
C05378=1094.024,-95.767,450.561,175.062,15.239,152.262
C05379=1094.030,-95.517,450.552,175.063,15.240,152.262
C05380=1094.036,-95.267,450.542,175.065,15.240,152.262
C05381=1094.042,-95.018,450.531,175.066,15.241,152.262
C05382=1094.048,-94.767,450.521,175.068,15.241,152.261
C05383=1094.055,-94.518,450.511,175.070,15.242,152.261
C05384=1094.060,-94.268,450.500,175.072,15.243,152.261
C05385=1094.067,-94.019,450.490,175.073,15.243,152.261
C05386=1094.072,-93.769,450.480,175.075,15.243,152.260
C05387=1094.078,-93.519,450.470,175.077,15.244,152.260
C05388=1094.084,-93.269,450.459,175.078,15.245,152.260
C05389=1094.090,-93.020,450.449,175.080,15.245,152.260
C05390=1094.096,-92.770,450.439,175.082,15.246,152.259
C05391=1094.102,-92.521,450.429,175.084,15.247,152.259
C05392=1094.108,-92.271,450.419,175.085,15.247,152.259
C05393=1094.114,-92.022,450.408,175.087,15.247,152.259
C05394=1094.120,-91.771,450.398,175.088,15.248,152.258
C05395=1094.127,-91.522,450.388,175.090,15.249,152.258
C05396=1094.132,-91.271,450.377,175.091,15.249,152.258
C05397=1094.139,-91.022,450.367,175.093,15.250,152.258
C05398=1094.144,-90.772,450.357,175.095,15.251,152.258
C05399=1094.150,-90.523,450.347,175.097,15.251,152.257
C05400=1094.156,-90.273,450.336,175.098,15.252,152.257
C05401=1094.162,-90.023,450.326,175.100,15.252,152.257
C05402=1094.169,-89.773,450.315,175.102,15.253,152.257
C05403=1094.174,-89.523,450.305,175.103,15.253,152.256
C05404=1094.181,-89.274,450.294,175.105,15.254,152.256
C05405=1094.186,-89.025,450.284,175.107,15.254,152.256
C05406=1094.193,-88.775,450.274,175.108,15.256,152.256
C05407=1094.198,-88.525,450.263,175.109,15.256,152.255
C05408=1094.204,-88.276,450.254,175.111,15.256,152.255
C05409=1094.211,-88.025,450.242,175.113,15.257,152.255
C05410=1094.217,-87.776,450.231,175.115,15.258,152.255
C05411=1094.223,-87.526,450.222,175.116,15.258,152.254
C05412=1094.228,-87.277,450.211,175.118,15.259,152.254
C05413=1094.235,-87.027,450.201,175.120,15.259,152.254
C05414=1094.241,-86.777,450.190,175.121,15.260,152.254
C05415=1094.247,-86.527,450.179,175.123,15.261,152.253
C05416=1094.253,-86.277,450.170,175.124,15.261,152.253
C05417=1094.259,-86.028,450.159,175.126,15.262,152.253
C05418=1094.265,-85.779,450.149,175.128,15.263,152.253
C05419=1094.271,-85.528,450.137,175.130,15.263,152.252
C05420=1094.277,-85.278,450.127,175.131,15.263,152.252
C05421=1094.283,-85.029,450.117,175.133,15.265,152.252
C05422=1094.289,-84.780,450.106,175.135,15.265,152.252
C05423=1094.295,-84.530,450.096,175.137,15.266,152.252
C05424=1094.302,-84.280,450.085,175.138,15.266,152.251
C05425=1094.307,-84.030,450.074,175.140,15.267,152.251
C05426=1094.314,-83.780,450.065,175.141,15.267,152.251
C05427=1094.319,-83.531,450.054,175.143,15.268,152.251
C05428=1094.326,-83.282,450.044,175.145,15.269,152.250
C05429=1094.332,-83.032,450.032,175.146,15.269,152.250
C05430=1094.338,-82.781,450.022,175.148,15.270,152.250
C05431=1094.344,-82.532,450.012,175.150,15.271,152.250
C05432=1094.350,-82.283,450.001,175.152,15.271,152.249
C05433=1094.356,-82.033,449.990,175.153,15.272,152.249
C05434=1094.363,-81.783,449.980,175.155,15.272,152.249
C05435=1094.368,-81.533,449.969,175.156,15.273,152.249
C05436=1094.374,-81.283,449.958,175.158,15.274,152.249
C05437=1094.380,-81.012,449.947,175.160,15.275,152.248
C05438=1094.388,-80.740,449.936,175.162,15.275,152.248
C05439=1094.394,-80.468,449.924,175.164,15.276,152.248
C05440=1094.401,-80.195,449.913,175.166,15.277,152.248
